# B&R Automation Studio project dbserv_0640 (part 19)

#### iodrv.c
```c
#ifdef _DEFAULT_INCLUDES
	#include <AsDefault.h>
#endif
/******************************************************************************
*    COPYRIGHT    BERNECKER + RAINER Industrie-Elektronik Ges.m.b.H           *
*******************************************************************************
*  Projekt:  I/O-Treiber
*  Teil:     Hauptprogramm
*  Datei:    iodrv.c
*  Typ:      GNU-C (32 Bit)
*------------------------------------------------------------------------------
*  Revision: 01.00
*  Datum:    05-04-2006
*  Autor:    WAI
*------------------------------------------------------------------------------
*  Funktion:
*------------------------------------------------------------------------------
*  Rev.  | Datum    | Name | Kommentar
*  ------+----------+------+---------------------------------------------------
*  01.00 | 05-04-06 | WAI  | Datei-Erstellung
*  01.01 | 26-11-10 | WAI  | Schreibzugriff auf PVs aktiviert
*        |          |      |
******************************************************************************/

/***********************************************************************/
/* Headerfiles einbinden                                               */
/***********************************************************************/

#include <bur\plc.h>			/* RPS-spezifische Typendeklarationen */
#include <string.h>
#include <dvframe.h>
#include <sys_lib.h>
#include <brsystem.h>
#include <fileio.h>
#include "iodrv.h"				/* globale Variablen und Konstanten */
#include "iodrv_parse.h"		/* Parser Funktionen */
#include "dbserv.h"				/* Meldeserver */

_LOCAL_RETAIN	BOOL	go	;
_LOCAL	UINT	LinkStat,SetStat,ScanStat,GetStat;

/***********************************************************************/
/* 					Initialisierungs-Unterprogramm                     */
/***********************************************************************/

void _INIT init_iodrv(void)
{

	int	item,i;
	IODRV_DP_Info_typ		*pIODRV_DP_Info;

	/*--------------------------------*/
	/* Variablen initialisieren       */
	/*--------------------------------*/
	for(i=0;i<ITEM_DIAGNOSE_SIZE;i++) {
		IODRV_ItemDiagnose[i].showData	= 0;
	}

	memset(&SYS_Statistic,0,sizeof(SYS_Statistic));

	myidBrServer			= 0;											/* ID BR-Server */

	rt_info.enable = 1; 													/* Taskklassenzykluszeit ermitteln */
	RTInfo(&rt_info);
	if(rt_info.status==0)	CycleTime	= (rt_info.cycle_time / 1000);		/* Zykluszeit in ms */
	else 					CycleTime	= 10;								/* Zykluszeit in ms */

	Error	= 0;															/* Generelle Variable fuer Initialisierungsfehler */

	initPAB = 1;

	/*****************************************************************************/
	/* Initialisierung nach Konfigurationsdatenmodul dplist und typlist (DbServ) */
	/*****************************************************************************/

	/*--------------------------------------------------*/
	/* Konfiguration aus Konfigurationsmodulen auslesen */
	/*--------------------------------------------------*/

	iodrv_parser();

	/* Kein Schwerwiegender Fehler beim Parsen */
	if(IODRV_ParserInfo.error==0) {
		/* für alle Items die PV suchen */
		for(item=0;item<IODRV_ParserInfo.NrOfItems;item++)	{
			pIODRV_DP_Info = (IODRV_DP_Info_typ *) (IODRV_ParserInfo.memAdr);
			pIODRV_DP_Info += item;

			if(pIODRV_DP_Info->DPNameLen && pIODRV_DP_Info->DPName !=NULL)	{
				/* PV-Namen aus DP- und Item-Namen zusammensetzen */
				strncpy(pIODRV_DP_Info->PVName,pIODRV_DP_Info->DPName,pIODRV_DP_Info->DPNameLen);
				if(pIODRV_DP_Info->ItemNameLen && pIODRV_DP_Info->ItemName !=NULL)	{
					strncat(pIODRV_DP_Info->PVName,pIODRV_DP_Info->ItemName,pIODRV_DP_Info->ItemNameLen);
				}
				/* PV-Adresse bestimmen */
				statePV_xgetadr = PV_xgetadr(pIODRV_DP_Info->PVName, &pIODRV_DP_Info->PVAdrs, &pIODRV_DP_Info->PVDataLen);
				if (statePV_xgetadr != 0) {
					/* Fehler PV */
						iodrv_parser_warn(PARS_ERR_PV_NOT_FOUND,"PV nicht vorhanden", pIODRV_DP_Info->PVName, 0,0, 0, 0, 0, 0);
				}
			}
		}
	}
}
/************************************************************************/
/* schreibt aktuellen Datenpunkt in das PAB 							*/
void WritePVtoPAB(IODRV_DP_Info_typ *pIODRV_DP_Info)
{
	int						do_it;
	PAR_TYPE				WertServer;
	UDINT					SizeServer;

	/* nur Lese- bzw. Schreib/Lese-Items an das PAB übergeben */
	if (myidBrServer == 0) {
		pIODRV_DP_Info->ErrorInfo = 2;				/* Info Server ID unbekannt */
	}
	else {
		pIODRV_DP_Info->AccessCounter += 1;			/* Zaehler inkrementieren: Signal wird an Server uebergeben */
		do_it = 1;

		switch(pIODRV_DP_Info->ItemTypNr) {
			case BOOL_IDX:
				pIODRV_DP_Info->ValueIO = *(BOOL *) pIODRV_DP_Info->PVAdrs;
				SizeServer  = sizeof(BOOL);
				if(pIODRV_DP_Info->Invers)	{
					WertServer.b	= (BOOL)pIODRV_DP_Info->ValueIO ^1;
				}
				else {
					WertServer.b	= (BOOL)pIODRV_DP_Info->ValueIO;
				}
				if(!initPAB && !WertServer.b && pIODRV_DP_Info->Quitt)	{
					do_it = 0;				/* gegangener, quittierpflichtiger DP nicht in PAB eintragen */
				}
				break;
			case USINT_IDX:
				WertServer.ui1	= *(USINT*)	pIODRV_DP_Info->PVAdrs;
				SizeServer  = sizeof(USINT);
				break;
			case SINT_IDX:
				WertServer.i1	= *(SINT*)	pIODRV_DP_Info->PVAdrs;
				SizeServer  = sizeof(SINT);
				break;
			case UINT_IDX:
				WertServer.ui2	= *(UINT*)	pIODRV_DP_Info->PVAdrs;
				SizeServer  = sizeof(UINT);
				break;
			case INT_IDX:
				WertServer.i2	= *(INT*)	pIODRV_DP_Info->PVAdrs;
				SizeServer  = sizeof(INT);
				break;
			case UDINT_IDX:
				WertServer.ui4	= *(UDINT*)	pIODRV_DP_Info->PVAdrs;
				SizeServer  = sizeof(UDINT);
				break;
			case DINT_IDX:
				WertServer.i4	= *(DINT*)	pIODRV_DP_Info->PVAdrs;
				SizeServer  = sizeof(DINT);
				break;
			default:
				WertServer.i2	= *(INT*)	pIODRV_DP_Info->PVAdrs;
				SizeServer  = sizeof(INT);
				break;
		}
		if(do_it)	{
			StatusSetValueItem = SetValueItem ((ACCESS_SERVER*)	myidBrServer,
												pIODRV_DP_Info->AnlagenNr,
												1,									/* Stationsnummer  immer 1 */
												pIODRV_DP_Info->DPTypNr,	  		/* Datenpunkttyp    */
												pIODRV_DP_Info->DPNr,			 	/* Datenpunktnummer */
												pIODRV_DP_Info->ItemNr,				/* Item */
												(USINT *) &WertServer,				/* Adresse Messwert */
												SizeServer,
												TimeBuf,
												0,			/* TimeStampNow=0 wegen Alarmliste, setze Zeitstempel bei Bedarf */
												1);
			if(!StatusSetValueItem)	{
				pIODRV_DP_Info->AccessCounter += 1;				/* Zaehler inkrementieren: Uebergabe an Server korrekt erfolgt */
				pIODRV_DP_Info->ErrorInfo		= 0;
			}
			else {
				pIODRV_DP_Info->ErrorInfo = 3;
			}
		}
	}
}

/***********************************************************************/
/* 						zyklisches Hauptprogramm                       */
/***********************************************************************/

void _CYCLIC cyclic_iodrv(void)
{
	int						item;
	IODRV_DP_Info_typ		*pIODRV_DP_Info;
	USINT	WriteBuffer[32];
	UDINT	len, lenTimeStamp;
	USINT	*pByteValue;

	/* Einlesen der Echtzeituhr */
	RTC_gettime(&TimeBuf);

	/* ID Meldeserver besorgen */
	get_idBrServer();

	if(go)	{
		go=0;
		iodrv_parser();

		/* Kein Schwerwiegender Fehler beim Parsen */
		if(IODRV_ParserInfo.error==0) {
			/* für alle Items die PV suchen */
			for(item=0;item<IODRV_ParserInfo.NrOfItems;item++)	{
				pIODRV_DP_Info = (IODRV_DP_Info_typ *) (IODRV_ParserInfo.memAdr);
				pIODRV_DP_Info += item;

				if(pIODRV_DP_Info->DPNameLen && pIODRV_DP_Info->DPName !=NULL)	{
					/* PV-Namen aus DP- und Item-Namen zusammensetzen */
					strncpy(pIODRV_DP_Info->PVName,pIODRV_DP_Info->DPName,pIODRV_DP_Info->DPNameLen);
					if(pIODRV_DP_Info->ItemNameLen && pIODRV_DP_Info->ItemName !=NULL)	{
						strncat(pIODRV_DP_Info->PVName,pIODRV_DP_Info->ItemName,pIODRV_DP_Info->ItemNameLen);
					}
					/* PV-Adresse bestimmen */
					statePV_xgetadr = PV_xgetadr(pIODRV_DP_Info->PVName, &pIODRV_DP_Info->PVAdrs, &pIODRV_DP_Info->PVDataLen);
					if (statePV_xgetadr != 0) {
						/* Fehler PV */
						iodrv_parser_warn(PARS_ERR_PV_NOT_FOUND,"PV nicht vorhanden", pIODRV_DP_Info->PVName, 0,0, 0, 0, 0, 0);
					}
				}
			}
		}
	}

	/* Diagnose */
	iodrv_mem_diagnose();

	/* -------------------------------*/
	/* Uebergabe an Server            */
	/* -------------------------------*/

	for(item=0;item<IODRV_ParserInfo.NrOfItems;item++)	{
		pIODRV_DP_Info = (IODRV_DP_Info_typ *) (IODRV_ParserInfo.memAdr);
		pIODRV_DP_Info += item;

		if(pIODRV_DP_Info->PVAdrs != NULL)	{
			if(pIODRV_DP_Info->Dir == cKW_READ)	{
				WritePVtoPAB(pIODRV_DP_Info);				/* PV ins PAB schreiben */
			}
			else if(pIODRV_DP_Info->Dir == cKW_READWRITE || pIODRV_DP_Info->Dir == cKW_WRITE)	{
				/* Item zum Schreiben anmelden */
				LinkStat = LinkWriteItem((ACCESS_SERVER*)myidBrServer, cINSTANCE_IODRV,
						pIODRV_DP_Info->AnlagenNr, 1, pIODRV_DP_Info->DPTypNr, pIODRV_DP_Info->DPNr, pIODRV_DP_Info->ItemNr,
						(UDINT)pIODRV_DP_Info);
				if (LinkStat != cEC_OK && LinkStat != cEC_ITEM_ALREADY_LINKED)	pIODRV_DP_Info->ErrorInfo = LinkStat;
				/* prüfen, ob Item geschrieben wurde */
				ScanStat = ScanWriteItem((ACCESS_SERVER*)myidBrServer, cINSTANCE_IODRV,
											WriteBuffer, sizeof(WriteBuffer),
											&len, &lenTimeStamp);
				if (ScanStat != cEC_OK)	pIODRV_DP_Info->ErrorInfo = ScanStat;
				if (ScanStat == cEC_OK) {
					/* für mich ? */
					GetStat = cEC_NO_DATA_IN_WRITEBUFFER;
					if (((WRITE_PIPE_DATA*)WriteBuffer)->pData == (unsigned char *)pIODRV_DP_Info) {
						GetStat = GetWriteItem((ACCESS_SERVER*)myidBrServer, cINSTANCE_IODRV,
												WriteBuffer, sizeof(WriteBuffer),
												&len, &lenTimeStamp);
						if (GetStat != cEC_OK)	pIODRV_DP_Info->ErrorInfo = GetStat;
						if (GetStat== cEC_OK) {
							if (((WRITE_PIPE_DATA*)WriteBuffer)->length == pIODRV_DP_Info->PVDataLen) {
								pByteValue = WriteBuffer + sizeof(WRITE_PIPE_DATA);
/* #if 0 26.11.10 Wai Kommentar entfernt */
								switch(pIODRV_DP_Info->ItemTypNr) {
									case BOOL_IDX:
										*(BOOL *)pIODRV_DP_Info->PVAdrs =  *(BOOL*)pByteValue;
										break;
									case USINT_IDX:
										*(USINT *)pIODRV_DP_Info->PVAdrs =  *(USINT*)pByteValue;
										break;
									case SINT_IDX:
										*(SINT *)pIODRV_DP_Info->PVAdrs =  *(SINT*)pByteValue;
										break;
									case UINT_IDX:
										*(UINT *)pIODRV_DP_Info->PVAdrs =  *(UINT*)pByteValue;
										break;
									case INT_IDX:
										*(INT *)pIODRV_DP_Info->PVAdrs =  *(INT*)pByteValue;
										break;
									case UDINT_IDX:
										*(UDINT *)pIODRV_DP_Info->PVAdrs =  *(UDINT*)pByteValue;
										break;
									case DINT_IDX:
										*(DINT *)pIODRV_DP_Info->PVAdrs =  *(DINT*)pByteValue;
										break;
								}
/* #endif 26.11.10 Wai Kommentar entfernt */

								/* Wert auch nach PAB zurückschreiben */
								SetStat = SetValueItem((ACCESS_SERVER*)myidBrServer,
										pIODRV_DP_Info->AnlagenNr, 1, pIODRV_DP_Info->DPTypNr, pIODRV_DP_Info->DPNr, pIODRV_DP_Info->ItemNr,
										pByteValue, sizeof(INT), TimeBuf, 0, TRUE);
								if (SetStat != cEC_OK)	pIODRV_DP_Info->ErrorInfo = SetStat;
							} /* (((WRITE_PIPE_DATA*)WriteBuffer)->length == PVDataLen */
							else {
								SetStat = cEC_INVALID_LENGTH;
								if (SetStat != cEC_OK)	pIODRV_DP_Info->ErrorInfo = SetStat;
							}
						} /* (intStat == cEC_OK) */
					} /* (((WRITE_PIPE_DATA*)WriteBuffer)->pData == (unsigned char*)inst->FubRef.this) */
				} /* (intStat == cEC_OK) */
				if (ScanStat != cEC_OK || GetStat != cEC_OK)	{
					/* keine Schreibdaten vorhanden: PV ins PAB schreiben */
					if(pIODRV_DP_Info->Dir == cKW_READWRITE)	{
						WritePVtoPAB(pIODRV_DP_Info);				/* PV ins PAB schreiben */
					}
				}
			} /* else if(pIODRV_DP_Info->Dir == cKW_READWRITE || pIODRV_DP_Info->Dir == cKW_WRITE)	*/
		} /* if(pIODRV_DP_Info->PVAdrs != NULL)	*/
	} /* for all Items */
	if(myidBrServer) initPAB = 0;

}

/*** eof *****************************************************************************/
```

#### iodrv_parse.c
```c
#ifdef _DEFAULT_INCLUDES
	#include <AsDefault.h>
#endif
/******************************************************************************
*    COPYRIGHT    BERNECKER + RAINER Industrie-Elektronik Ges.m.b.H           *
*******************************************************************************
*  Projekt:  I/O-Treiber
*  Teil:     Parserfunktionen
*  Datei:    iodrv_parse.c
*  Typ:      GNU-C (32 Bit)
*------------------------------------------------------------------------------
*  Revision: 01.00
*  Datum:    05-04-2006
*  Autor:    WAI
*------------------------------------------------------------------------------
*  Funktion:
*------------------------------------------------------------------------------
*  Rev.  | Datum    | Name | Kommentar
*  ------+----------+------+---------------------------------------------------
*  01.00 | 05-04-06 | WAI  | Datei-Erstellung
*  02.00 | 10-07-26 | BIE  | strnicmp gegen strncasecmp ersetzt
*        |          |      |
******************************************************************************/
#include <bur\plc.h>			/* RPS-spezifische Typendeklarationen */
#include <string.h>
#include <dvframe.h>
#include <sys_lib.h>
#include <asbrstr.h>
#include <brsystem.h>
#include "iodrv.h"
#include "iodrv_parse.h"
#include "parser.h"

/**********************************************************
*		Konfiguration aus Datenmodul auslesen
**********************************************************/
void iodrv_parser()
{
	plcbit				BlockFound,DPFound,TypFound,ItemFound;
	IODRV_DP_Info_typ		*pIODRV_DP_Info;
	unsigned char ANr[20];

	memset(&IODRV_ParserInfo,0,sizeof(IODRV_ParserInfo));
	IODRV_ParserInfo.ErrorMsg = 1;									/* Freigabe: Fehlermeldungen ins Logbuch eintragen */

	/*--------------------------------------------------*/
	/* Info ueber Datenmodul dplist und typlist besorgen*/
	/*--------------------------------------------------*/

	DOI_dplist.enable	= 1;
	DOI_dplist.pName	= (unsigned long) DATA_OBJEKT_DPLIST;
	DatObjInfo((DatObjInfo_typ*) &DOI_dplist);

	DOI_typlist.enable	= 1;
	DOI_typlist.pName	= (unsigned long) DATA_OBJEKT_TYPLIST;
	DatObjInfo((DatObjInfo_typ*) &DOI_typlist);

	/*--------------------------------------------------*/
	/* Fehlermeldung: Datenmodul dplist nicht vorhanden */
	/*--------------------------------------------------*/
	if(DOI_typlist.status) {
		iodrv_parser_err(PARS_ERR_DPLIST_NOT_FOUND, "Datenmodul fehlt:", (unsigned char *) DOI_dplist.pName, 0, 0, 0, 0, 0, 0);
	}

	/*--------------------------------------------------*/
	/* Fehlermeldung: Datenmodul typlist nicht vorhanden */
	/*--------------------------------------------------*/
	if(DOI_typlist.status) {
		iodrv_parser_err(PARS_ERR_TYPLIST_NOT_FOUND, "Datenmodul fehlt:", (unsigned char *) DOI_typlist.pName, 0, 0, 0, 0, 0, 0);
	}

	/*--------------------------------------------------*/
	/* Globale Parameter lesen							*/
	/*--------------------------------------------------*/
	if(!IODRV_ParserInfo.error) {

		iodrv_parser_dplist_clear();									/* Parsen von Beginn an */

		memset(&IODRV_GlobalData,0,sizeof(IODRV_GlobalData));			/* Parameterstruktur loeschen */

		iodrv_parser_global();											/* Parameter parsen */
	}

	/*------------------------------------------------------*/
	/* Anzahl Datenpunkte und Items ermitteln				*/
	/*------------------------------------------------------*/

	if(!IODRV_ParserInfo.error) {

		IODRV_ParserInfo.ErrorMsg = 0;															/* Keine Eintrage ins Logbuch */
		iodrv_parser_dplist_clear();															/* dplist von Beginn an Parsen */
		memset(&IODRV_BlockData,0,sizeof(IODRV_BlockData));										/* Info ueber Blockparameter loeschen */

		do {
			memset(&IODRV_DPData,0,sizeof(IODRV_DPData));											/* Info ueber Datenpunkt loeschen */
			copyItemData((IODRV_ItemData_typ *) &IODRV_DPData,(IODRV_ItemData_typ *) &IODRV_BlockData);	/* Blockparameter uebernehmen */

			BlockFound	= 0;
			DPFound		= 0;

			iodrv_parser_dpinfo((plcbit *) &BlockFound,(plcbit *) &DPFound);						/* Nächsten Datenpunkt für IODRV-Treiber suchen */

			if(DPFound) {																	/* Datenpunkt für IODRV-Treiber gefunden */
				IODRV_ParserInfo.NrOfDataPoints++;											/* Anzahl Datenpunkte pro Linie zählen */
				if(IODRV_DPData.Typ.defined) {												/* Ist zu dem Datenpunkt der Datentyp definiert ? */
					iodrv_parser_typlist_clear();											/* typlist von Beginn an Parsen */
					TypFound = iodrv_parser_dptype(IODRV_DPData.Typ.name, IODRV_DPData.Typ.size); /* Datentyp in typlist suchen */
					if(TypFound) {															/* Datentyp wurde in typlist gefunden */
						/* Anzahl Items des Datenpunktes ermitteln */
						do {
							memset(&IODRV_ItemData,0,sizeof(IODRV_ItemData));				/* Struktur für ITEM-Parameter loeschen */
							ItemFound = iodrv_parser_iteminfo();							/* Item in typlist suchen */
							if(ItemFound) {													/* Item wurde gefunden */
								copyItemData((IODRV_ItemData_typ *) &IODRV_ItemData,(IODRV_ItemData_typ *) &IODRV_DPData);
								IODRV_ParserInfo.NrOfItems++;								/* Anzahl der Items ermitteln */
							}
						} while(ItemFound);

					} /* if(TypFound) */
				} /* if(IODRV_DPData.Typ.defined) */
			} /* if(DPFound) */
		} while(DPFound || BlockFound);
	} /* if(!IODRV_ParserInfo.error) */

	/*------------------------------------------------------*/
	/* Speicher fuer alle Items allokieren					*/
	/*------------------------------------------------------*/

	if(!IODRV_ParserInfo.error) {
		IODRV_ParserInfo.ErrorMsg	= 1;					/* Freigabe: Fehlermeldungen ins Logbuch eintragen */
		IODRV_ParserInfo.memSize = IODRV_ParserInfo.NrOfItems * sizeof(IODRV_DP_Info_typ);
		IODRV_ParserInfo.allocStatus = TMP_alloc(IODRV_ParserInfo.memSize, (void**) &IODRV_ParserInfo.memAdr); 	/* allocate new memory from RAM*/
		if(IODRV_ParserInfo.allocStatus) {
			iodrv_parser_err(PARS_ERR_MEM_ALLOC, "Fehler TMP_alloc:", 0, "Groesse:", IODRV_ParserInfo.memSize, "Status:", (long) IODRV_ParserInfo.allocStatus, 0, 0);
		}
		else {
			memset((void *) IODRV_ParserInfo.memAdr,0,IODRV_ParserInfo.memSize);
		}
	}

	/*-----------------------------------------------------------------------*/
	/* Iteminformationen auslesen und in Speicher eintragen     */
	/*-----------------------------------------------------------------------*/

	if(!IODRV_ParserInfo.error) {

		iodrv_parser_dplist_clear();																/* dplist von Beginn an Parsen */
		memset(&IODRV_BlockData,0,sizeof(IODRV_BlockData));											/* Info ueber Blockparameter loeschen */

		do {
			memset(&IODRV_DPData,0,sizeof(IODRV_DPData));											/* Info ueber Datenpunkt loeschen */
			copyItemData((IODRV_ItemData_typ *) &IODRV_DPData,(IODRV_ItemData_typ *) &IODRV_BlockData);	/* Blockparameter uebernehmen */
			BlockFound	= 0;
			DPFound		= 0;
			iodrv_parser_dpinfo((plcbit *) &BlockFound,(plcbit *) &DPFound);						/* Nächsten Datenpunkt für IODRV-Treiber suchen */
			if(DPFound) {																		/* Datenpunkt für IODRV-Treiber gefunden */
				if(iodrv_parser_dpinfo_ok((IODRV_ItemData_typ *) &IODRV_DPData)) {					/* Alle notwendigen Angaben vorhanden und korrekt ? */
																								/* Zugehoerigen Linienindex suchen */
					iodrv_parser_typlist_clear();												/* typlist von Beginn an Parsen */
					TypFound = iodrv_parser_dptype(IODRV_DPData.Typ.name, IODRV_DPData.Typ.size); /* Datentyp in typlist suchen */
					if(TypFound) {															/* Datentyp wurde in typlist gefunden */
						/* Anzahl Items des Datenpunktes ermitteln */
						do {
							memset(&IODRV_ItemData,0,sizeof(IODRV_ItemData));					/* Struktur für ITEM-Parameter loeschen */
																								/* Parameter des Datenpunktes auf Item übertragen */
							copyItemData((IODRV_ItemData_typ *) &IODRV_ItemData,(IODRV_ItemData_typ *) &IODRV_DPData);

							ItemFound = iodrv_parser_iteminfo();								/* Item in typlist suchen */
							if(ItemFound) {													/* Item wurde gefunden */

																							/* Pruefen, ob Parameter vollstaendig und korrekt sind */
								if(iodrv_parser_iteminfo_ok((IODRV_ItemData_typ *) &IODRV_ItemData)) {
									pIODRV_DP_Info = (IODRV_DP_Info_typ *) (IODRV_ParserInfo.memAdr);
									pIODRV_DP_Info += IODRV_ParserInfo.ActItemIdx;

																						/* Daten in Speicher eintragen */
									pIODRV_DP_Info->AnlagenNr	= (UINT)	IODRV_ItemData.AnlagenNr.value;
									pIODRV_DP_Info->DPNr		= (UINT)	IODRV_ItemData.DPNr.value;
									pIODRV_DP_Info->DPTypNr		= (UINT)	IODRV_ItemData.DPTypNr.value;
									pIODRV_DP_Info->DPName		= (USINT *)	IODRV_ItemData.DPName.name;
									pIODRV_DP_Info->DPNameLen	= (UINT)	IODRV_ItemData.DPName.size;
									pIODRV_DP_Info->ItemNr		= (UINT)	IODRV_ItemData.ItemNr.value;
									pIODRV_DP_Info->ItemTypNr	= (USINT)	IODRV_ItemData.ItemTypNr.value;
									pIODRV_DP_Info->ItemName	= (USINT *)	IODRV_ItemData.ItemName.name;
									pIODRV_DP_Info->ItemNameLen	= (UINT)	IODRV_ItemData.ItemName.size;
									pIODRV_DP_Info->Invers		= (USINT)	IODRV_ItemData.Invers.value;
									pIODRV_DP_Info->Quitt		= (USINT)	IODRV_ItemData.Quitt.value;
									pIODRV_DP_Info->Dir			= (USINT)	IODRV_ItemData.Dir.value;

									IODRV_ParserInfo.ActItemIdx++;
								} /* if(!error) */
							} /* if(!error) */
						} while(ItemFound);
					} /* if(TypFound) */
				} /* if(iodrv_parser_dpinfo_ok())*/
			} /* if(DPFound) */
		} while(DPFound || BlockFound);
	} /* if(!IODRV_ParserInfo.error) */

	strcpy(MsgTxt,ERR_MSG_PRE_STRG);
	strcat(MsgTxt," Parser beendet");
	ERRxwarning( 0, bin_to_bcd_8(0),MsgTxt);

	strcpy(MsgTxt,ERR_MSG_PRE_STRG);
	strcat(MsgTxt," Anzahl Meldungen ");
	brsitoa(IODRV_ParserInfo.NrOfLogEntrys, (UDINT) &ANr);
	strcat(MsgTxt,ANr);
	ERRxwarning( 0, bin_to_bcd_8((unsigned long) IODRV_ParserInfo.NrOfLogEntrys), MsgTxt);

}

/**********************************************************
*		Globale Parameter aus Datennmodul lesen
**********************************************************/
void iodrv_parser_global()
{

	BOOL			dataReady;

		/* ----------------------------------------- */
	 	/* Globale Eintraege fuer IODRV-Treiber parsen */
		/* ----------------------------------------- */

		/* Parser-Status loeschen */
		State_find_StationTypPoint	= 0;
		State_find_Section			= 0;
		State_find_Data				= 0;

		while (PaDPList.pParser < (unsigned char*) DOI_dplist.pDatObjMem + DOI_dplist.len) {

			/* Suche nach Stations/Typ/Punkt-Beschreibung */
			State_find_StationTypPoint = find_StationTypPoint (	(unsigned char*) DOI_dplist.pDatObjMem, PaDPList.pParser,
																(unsigned char*) DOI_dplist.pDatObjMem + DOI_dplist.len,
																&PaDPList.pParser, &PaDPList.pParserLine, &PaDPList.pParserErr, &PaDPList.CountLines,
																&PaDPList.pDataArg1, &PaDPList.SizeArg1,
																&PaDPList.pDataArg2, &PaDPList.SizeArg2,
																&PaDPList.SectionType);
			/* keine Daten oder Fehler aufgetreten ? */
			if (State_find_StationTypPoint < 0) {
				break;
			}

			/* Pointer auf Station/Typ/Punkt */
			switch (PaDPList.SectionType) {

				/* ------------------ */
				/* Stations-Abschnitt */
				/* ------------------ */
				case cCD_STATION:
					do {
						State_find_Section = find_Section (
							(unsigned char*) DOI_dplist.pDatObjMem, PaDPList.pParser,
															(unsigned char*) DOI_dplist.pDatObjMem + DOI_dplist.len,
															&PaDPList.pParser, &PaDPList.pParserLine, &PaDPList.pParserErr, &PaDPList.CountLines,
															&PaDPList.pDataArg1, &PaDPList.SizeArg1,
															&PaDPList.pDataArg2, &PaDPList.SizeArg2,
															KW_IODRV_SECTION);

						/* keine Daten oder Fehler aufgetreten ? */
						if (State_find_Section < 0) {
							break;
						}

						/* Pointer auf Anfang der Sektion stellen */
						if (PaDPList.pDataArg2 != NULL) {
							PaDPList.pParser = PaDPList.pDataArg2;
						}
						else {
							continue;
						}

						/* alle Daten der Sektion bearbeiten */
						dataReady	= 0;
						do {
							/* Daten der Sektion anfordern */
							State_find_Data = find_Data (	(unsigned char*) DOI_dplist.pDatObjMem, PaDPList.pParser,
															(unsigned char*) DOI_dplist.pDatObjMem + DOI_dplist.len,
															  &PaDPList.pParser, &PaDPList.pParserLine, &PaDPList.pParserErr, NULL,
															  &PaDPList.pDataArg1, &PaDPList.SizeArg1,
															  &PaDPList.pDataArg2, &PaDPList.SizeArg2,
															  &PaDPList.pDataArg3, &PaDPList.SizeArg3);

							/* Zeilenende erreicht */
							if (State_find_Data == -1) {
								PaDPList.pParser++;
							}
							/* Daten vorhanden */
							else if (State_find_Data == TRUE) {
								/* noch keine globalen Daten vorhanden */
								if (0) {
								}
								/* Unbekannter Eintrag */
								else {
									iodrv_parser_warn(PARS_ERR_UNKNOWN_GLOBAL_ENTRY,"Eintrag unbekannt:", PaDPList.pParserLine, " / Zeile =", (long) PaDPList.CountLines, 0, 0, 0, 0);
								}
							}

							/* Endebedinung der Schleife: Keine Daten mehr vorhanden, oder Ende des Datenmodules erreicht */
							if((State_find_Data!=TRUE) && (State_find_Data!=-1))					dataReady = 1;
							if(PaDPList.pParser >= (unsigned char*) DOI_dplist.pDatObjMem + DOI_dplist.len)	dataReady = 1;
						} while (!dataReady);
					} while (State_find_Section == TRUE);
					break;
				case cCD_TYP:
					break;
				case cCD_POINT:
					break;
			}
		}
}

/*****************************************************************
*		Informationen ueber einen Datenpunkt ermitteln
******************************************************************/
void iodrv_parser_dpinfo(plcbit *pBlockFound, plcbit *pDPFound)
{

		*pDPFound	= 0;
		*pBlockFound= 0;

		/* -------------------------------------------- */
	 	/* Datenpunkt Eintraege fuer IODRV-Treiber parsen */
		/* -------------------------------------------- */

		/* Parser-Status loeschen */
		State_find_StationTypPoint	= 0;
		State_find_Section			= 0;
		State_find_Data				= 0;

		while (!*pDPFound && !*pBlockFound && (PaDPList.pParser < (unsigned char*) DOI_dplist.pDatObjMem + DOI_dplist.len)) {

			/* Suche nach Stations/Typ/Punkt-Beschreibung */
			State_find_StationTypPoint = find_StationTypPoint (	(unsigned char*) DOI_dplist.pDatObjMem, PaDPList.pParser,
																(unsigned char*) DOI_dplist.pDatObjMem + DOI_dplist.len,
																&PaDPList.pParser, &PaDPList.pParserLine, &PaDPList.pParserErr, &PaDPList.CountLines,
																&PaDPList.pDataArg1, &PaDPList.SizeArg1,
																&PaDPList.pDataArg2, &PaDPList.SizeArg2,
																&PaDPList.SectionType);
			/* keine Daten oder Fehler aufgetreten ? */
			if (State_find_StationTypPoint < 0) {
				break;
			}

			/* Pointer auf Station/Typ/Punkt */
			switch (PaDPList.SectionType) {
				/* ------------------ */
				/* Datentyp-Abschnitt */
				/* ------------------ */
				case cCD_POINT:

					/* Parserposition zwischenspeichern */
					memcpy(&PaDPListSave,&PaDPList,sizeof(PaDPListSave));

					pPointName = PaDPList.pDataArg1, lenPointName = PaDPList.SizeArg1;

					/* Suchen nach Sektion "IODRV" */
					do {
						State_find_Section = find_Section (	(unsigned char*) DOI_dplist.pDatObjMem, PaDPList.pParser,
															(unsigned char*) DOI_dplist.pDatObjMem + DOI_dplist.len,
															&PaDPList.pParser, 	 &PaDPList.pParserLine, &PaDPList.pParserErr, &PaDPList.CountLines,
															&PaDPList.pDataArg1, &PaDPList.SizeArg1,
															&PaDPList.pDataArg2, &PaDPList.SizeArg2,
															KW_IODRV_SECTION);

						/* keine Daten oder Fehler aufgetreten ? */
						if (State_find_Section < 0) {
							break;
						}

						/* Pointer auf Anfang der Sektion stellen */
						if (PaDPList.pDataArg2 != NULL) {
							PaDPList.pParser = PaDPList.pDataArg2;
						}
						else {
							continue;
						}

						/* alle Daten der Sektion bearbeiten */

						IODRV_DPData.DPName.name = pPointName;
						IODRV_DPData.DPName.size = lenPointName;
						IODRV_DPData.DPName.defined = 1;

						*pDPFound		= 1;
						iodrv_parser_data((unsigned char*) DOI_dplist.pDatObjMem,
										(unsigned char*) DOI_dplist.pDatObjMem + DOI_dplist.len,
										(Parser_typ *) &PaDPList,
										(IODRV_ItemData_typ *) &IODRV_DPData,
										IODRV_SECTION,DP_PART);

					} while (State_find_Section == TRUE);

					/* Parserposition rückholen */
					memcpy(&PaDPList,&PaDPListSave,sizeof(PaDPList));

					/* Suchen nach Sektion "ALL" */
					do {
						State_find_Section = find_Section (	(unsigned char*) DOI_dplist.pDatObjMem, PaDPList.pParser,
															(unsigned char*) DOI_dplist.pDatObjMem + DOI_dplist.len,
															&PaDPList.pParser, &PaDPList.pParserLine, &PaDPList.pParserErr, &PaDPList.CountLines,
															&PaDPList.pDataArg1, &PaDPList.SizeArg1,
															&PaDPList.pDataArg2, &PaDPList.SizeArg2,
															KW_ALL_SECTION);

						/* keine Daten oder Fehler aufgetreten ? */
						if (State_find_Section < 0) {
							break;
						}

						/* Pointer auf Anfang der Sektion stellen */
						if (PaDPList.pDataArg2 != NULL) {
							PaDPList.pParser = PaDPList.pDataArg2;
						}
						else {
							continue;
						}

						/* alle Daten der Sektion bearbeiten */
						iodrv_parser_data((unsigned char*) DOI_dplist.pDatObjMem,
										(unsigned char*) DOI_dplist.pDatObjMem + DOI_dplist.len,
										(Parser_typ *) &PaDPList,
										(IODRV_ItemData_typ *) &IODRV_DPData,
										ALL_SECTION,DP_PART);

					} while (State_find_Section == TRUE);
					break;

				/* ------------------ */
				/* Block-Abschnitt    */
				/* ------------------ */
				case cCD_TYP:
					if(strncasecmp(PaDPList.pDataArg1, KW_BLOCK_SECTION, PaDPList.SizeArg1) == 0 && strlen(KW_BLOCK_SECTION) == PaDPList.SizeArg1 ) {
						*pBlockFound = 1;

						/* Parserposition zwischenspeichern */
						memcpy(&PaDPListSave,&PaDPList,sizeof(PaDPListSave));

						/* Suchen nach Sektion "IODRV" */
						do {
							State_find_Section = find_Section (	(unsigned char*) DOI_dplist.pDatObjMem, PaDPList.pParser,
																(unsigned char*) DOI_dplist.pDatObjMem + DOI_dplist.len,
																&PaDPList.pParser, 	 &PaDPList.pParserLine, &PaDPList.pParserErr, &PaDPList.CountLines,
																&PaDPList.pDataArg1, &PaDPList.SizeArg1,
																&PaDPList.pDataArg2, &PaDPList.SizeArg2,
																KW_IODRV_SECTION);

							/* keine Daten oder Fehler aufgetreten ? */
							if (State_find_Section < 0) {
								break;
							}

							/* Pointer auf Anfang der Sektion stellen */
							if (PaDPList.pDataArg2 != NULL) {
								PaDPList.pParser = PaDPList.pDataArg2;
							}
							else {
								continue;
							}

							/* alle Daten der Sektion bearbeiten */

							iodrv_parser_data((unsigned char*) DOI_dplist.pDatObjMem,
											(unsigned char*) DOI_dplist.pDatObjMem + DOI_dplist.len,
											(Parser_typ *) &PaDPList,
											(IODRV_ItemData_typ *) &IODRV_BlockData,
											IODRV_SECTION,DP_PART);

						} while (State_find_Section == TRUE);

						/* Parserposition rückholen */
						memcpy(&PaDPList,&PaDPListSave,sizeof(PaDPList));

						/* Suchen nach Sektion "ALL" */
						do {
							State_find_Section = find_Section (	(unsigned char*) DOI_dplist.pDatObjMem, PaDPList.pParser,
																(unsigned char*) DOI_dplist.pDatObjMem + DOI_dplist.len,
																&PaDPList.pParser, &PaDPList.pParserLine, &PaDPList.pParserErr, &PaDPList.CountLines,
																&PaDPList.pDataArg1, &PaDPList.SizeArg1,
																&PaDPList.pDataArg2, &PaDPList.SizeArg2,
																KW_ALL_SECTION);

							/* keine Daten oder Fehler aufgetreten ? */
							if (State_find_Section < 0) {
								break;
							}

							/* Pointer auf Anfang der Sektion stellen */
							if (PaDPList.pDataArg2 != NULL) {
								PaDPList.pParser = PaDPList.pDataArg2;
							}
							else {
								continue;
							}

							/* alle Daten der Sektion bearbeiten */
							iodrv_parser_data((unsigned char*) DOI_dplist.pDatObjMem,
											(unsigned char*) DOI_dplist.pDatObjMem + DOI_dplist.len,
											(Parser_typ *) &PaDPList,
											(IODRV_ItemData_typ *) &IODRV_BlockData,
											ALL_SECTION,DP_PART);

						} while (State_find_Section == TRUE);
					}
					break;

			}
		}
}

/*****************************************************************
*		Datentyp in typlist suchen
******************************************************************/
plcbit iodrv_parser_dptype(unsigned char *pName, unsigned short size)
{

		BOOL	TypFound=0;

		/* -------------------------------------------- */
	 	/* Datenpunkt Eintraege fuer IODRV-Treiber parsen */
		/* -------------------------------------------- */

		/* Parser-Status loeschen */
		State_find_StationTypPoint	= 0;
		State_find_Section			= 0;
		State_find_Data				= 0;

		while (!TypFound && (PaTypList.pParser < (unsigned char*) DOI_typlist.pDatObjMem + DOI_typlist.len) && (State_find_StationTypPoint>=0)) {

			/* Suche nach Stations/Typ/Punkt-Beschreibung */
			State_find_StationTypPoint = find_StationTypPoint (	(unsigned char*) DOI_typlist.pDatObjMem, PaTypList.pParser,
																(unsigned char*) DOI_typlist.pDatObjMem + DOI_typlist.len,
																&PaTypList.pParser, &PaTypList.pParserLine, &PaTypList.pParserErr, &PaTypList.CountLines,
																&PaTypList.pDataArg1, &PaTypList.SizeArg1,
																&PaTypList.pDataArg2, &PaTypList.SizeArg2,
																&PaTypList.SectionType);
			/* keine Daten oder Fehler aufgetreten ? */
			if (State_find_StationTypPoint < 0) {
				break;
			}

			if(PaTypList.SectionType==cCD_TYP) {
				if((PaTypList.SizeArg1==size) && (strncasecmp(PaTypList.pDataArg1, pName, PaTypList.SizeArg1) == 0)) {
					TypFound = 1;

					/* Parserposition zwischenspeichern */
					memcpy(&PaTypListSave,&PaTypList,sizeof(PaTypListSave));

					/* Suchen nach Sektion "IODRV" */
					State_find_Section = find_Section (	(unsigned char*) DOI_typlist.pDatObjMem, PaTypList.pParser,
														(unsigned char*) DOI_typlist.pDatObjMem + DOI_typlist.len,
														&PaTypList.pParser, &PaTypList.pParserLine, &PaTypList.pParserErr, &PaTypList.CountLines,
														&PaTypList.pDataArg1, &PaTypList.SizeArg1,
														&PaTypList.pDataArg2, &PaTypList.SizeArg2,
														KW_IODRV_SECTION);

					/* Section gefunden ? Daten parsen */
					if (State_find_Section == TRUE) {

						/* Pointer auf Anfang der Sektion stellen */
						if (PaTypList.pDataArg2 != NULL) {
							PaTypList.pParser = PaTypList.pDataArg2;
						}
						else {
							continue;
						}

						iodrv_parser_data((unsigned char*) DOI_typlist.pDatObjMem,
										(unsigned char*) DOI_typlist.pDatObjMem + DOI_typlist.len,
										(Parser_typ *) &PaTypList,
										(IODRV_ItemData_typ *) &IODRV_DPData,
										IODRV_SECTION,DP_PART);
					}
					/* Parserposition rückkopieren */
					memcpy(&PaTypList,&PaTypListSave,sizeof(PaTypList));

					/* Suchen nach Sektion "ALL" */
					State_find_Section = find_Section (	(unsigned char*) DOI_typlist.pDatObjMem, PaTypList.pParser,
														(unsigned char*) DOI_typlist.pDatObjMem + DOI_typlist.len,
														&PaTypList.pParser, &PaTypList.pParserLine, &PaTypList.pParserErr, &PaTypList.CountLines,
														&PaTypList.pDataArg1, &PaTypList.SizeArg1,
														&PaTypList.pDataArg2, &PaTypList.SizeArg2,
														KW_ALL_SECTION);

					/* Section gefunden ? Daten parsen */
					if (State_find_Section == TRUE) {

						/* Pointer auf Anfang der Sektion stellen */
						if (PaTypList.pDataArg2 != NULL) {
							PaTypList.pParser = PaTypList.pDataArg2;
						}
						else {
							continue;
						}

						iodrv_parser_data((unsigned char*) DOI_typlist.pDatObjMem,
										(unsigned char*) DOI_typlist.pDatObjMem + DOI_typlist.len,
										(Parser_typ *) &PaTypList,
										(IODRV_ItemData_typ *) &IODRV_DPData,
										ALL_SECTION,DP_PART);
					}
					/* Parserposition rückkopieren */
					memcpy(&PaTypList,&PaTypListSave,sizeof(PaTypList));

				}
			}
		}
	return(TypFound);
}

/*****************************************************************
*		Informationen ueber ein Item ermitteln
******************************************************************/
plcbit iodrv_parser_iteminfo()
{

		BOOL	ItemFound=0;

		/* -------------------------------------------- */
	 	/* Datenpunkt Eintraege fuer IODRV-Treiber parsen */
		/* -------------------------------------------- */

		/* Parser-Status loeschen */
		State_find_StationTypPoint	= 0;
		State_find_Section			= 0;
		State_find_Data				= 0;

		while (!ItemFound && (PaTypList.pParser < (unsigned char*) DOI_typlist.pDatObjMem + DOI_typlist.len)) {

			/* Suche nach Stations/Typ/Punkt-Beschreibung */
			State_find_StationTypPoint = find_StationTypPoint (	(unsigned char*) DOI_typlist.pDatObjMem, PaTypList.pParser,
																(unsigned char*) DOI_typlist.pDatObjMem + DOI_typlist.len,
																&PaTypList.pParser, &PaTypList.pParserLine, &PaTypList.pParserErr, &PaTypList.CountLines,
																&PaTypList.pDataArg1, &PaTypList.SizeArg1,
																&PaTypList.pDataArg2, &PaTypList.SizeArg2,
																&PaTypList.SectionType);
			/* keine Daten oder Fehler aufgetreten ? */
			if (State_find_StationTypPoint < 0) {
				break;
			}

			if(PaTypList.SectionType==cCD_ITEM) {

				/* Parserposition zwischenspeichern */
				memcpy(&PaTypListSave,&PaTypList,sizeof(PaTypListSave));

				/* Suchen nach Sektion "IODRV" */
				State_find_Section = find_Section (	(unsigned char*) DOI_typlist.pDatObjMem, PaTypList.pParser,
													(unsigned char*) DOI_typlist.pDatObjMem + DOI_typlist.len,
													&PaTypList.pParser, &PaTypList.pParserLine, &PaTypList.pParserErr, &PaTypList.CountLines,
													&PaTypList.pDataArg1, &PaTypList.SizeArg1,
													&PaTypList.pDataArg2, &PaTypList.SizeArg2,
													KW_IODRV_SECTION);

				/* keine Daten oder Fehler aufgetreten ? */
				if (State_find_Section < 0) {
					break;
				}

				/* Pointer auf Anfang der Sektion stellen */
				if (PaTypList.pDataArg2 != NULL) {
					PaTypList.pParser = PaTypList.pDataArg2;
				}
				else {
					continue;
				}

				ItemFound	= 1;

				iodrv_parser_data((unsigned char*) DOI_typlist.pDatObjMem,
								(unsigned char*) DOI_typlist.pDatObjMem + DOI_typlist.len,
								(Parser_typ *) &PaTypList,
								(IODRV_ItemData_typ *) &IODRV_ItemData,
								IODRV_SECTION,ITEM_PART);

				/* Parserposition rückkopieren */
				memcpy(&PaTypList,&PaTypListSave,sizeof(PaTypList));

				/* Suchen nach Sektion "ALL" */
				State_find_Section = find_Section (	(unsigned char*) DOI_typlist.pDatObjMem, PaTypList.pParser,
													(unsigned char*) DOI_typlist.pDatObjMem + DOI_typlist.len,
													&PaTypList.pParser, &PaTypList.pParserLine, &PaTypList.pParserErr, &PaTypList.CountLines,
													&PaTypList.pDataArg1, &PaTypList.SizeArg1,
													&PaTypList.pDataArg2, &PaTypList.SizeArg2,
													KW_ALL_SECTION);

				/* keine Daten oder Fehler aufgetreten ? */

				if (State_find_Section>0) {

					/* Pointer auf Anfang der Sektion stellen */
					if (PaTypList.pDataArg2 != NULL) {
						PaTypList.pParser = PaTypList.pDataArg2;
					}
					else {
						continue;
					}

					iodrv_parser_data((unsigned char*) DOI_typlist.pDatObjMem,
									(unsigned char*) DOI_typlist.pDatObjMem + DOI_typlist.len,
									(Parser_typ *) &PaTypList,
									(IODRV_ItemData_typ *) &IODRV_ItemData,
									ALL_SECTION,ITEM_PART);

				}
			}
			else {
				break;
			}

		}

	return(ItemFound);
}

/*****************************************************************
*	Datenbereich einer Sektion parsen
******************************************************************/
void iodrv_parser_data(unsigned char *pSrcStart,unsigned char *pSrcEnd, Parser_typ *pPa, IODRV_ItemData_typ *pData, unsigned char SectionInfo, unsigned char PartInfo) {

	plcbit			dataReady = 0;
	plcbit			dataFound = 0;
	unsigned char	Arg3IsANumber;
	long			Arg3Value;

	do {
		/* Daten der Sektion anfordern */
		State_find_Data = find_Data (	pSrcStart, pPa->pParser, pSrcEnd,
										  &pPa->pParser, &pPa->pParserLine, &pPa->pParserErr, NULL,
										  &pPa->pDataArg1, &pPa->SizeArg1,
										  &pPa->pDataArg2, &pPa->SizeArg2,
										  &pPa->pDataArg3, &pPa->SizeArg3);

		/* Zeilenende erreicht */
		if (State_find_Data == -1) {
			pPa->pParser++;
		}
		/* Daten vorhanden */
		else if (State_find_Data == TRUE) {

			dataFound = 0;

			/* Pruefen, ob Argument 3 einer Zahl entspricht */
			if(pPa->pDataArg3 != NULL && pPa->SizeArg3 != 0) {
				Arg3IsANumber	= IsANumber(pPa->pDataArg3);
				if(Arg3IsANumber==TRUE)	Arg3Value	= brsatoi((UDINT) pPa->pDataArg3);
			}
			else {
				Arg3IsANumber = FALSE;
			}

			/* Schlüsselworte pruefen, die nur im allgemeinen Datenpunktbereich vorkommen */
			if(PartInfo==DP_PART) {
				/* Anlagennummer */
				if (strncasecmp(pPa->pDataArg1, KW_DP_ALL_ANL, pPa->SizeArg1) == 0 && strlen(KW_DP_ALL_ANL) == pPa->SizeArg1 &&
					strncasecmp(pPa->pDataArg2, KW_DP_ALL_ANL_NR, pPa->SizeArg2) == 0 && strlen(KW_DP_ALL_ANL_NR) == pPa->SizeArg2 &&
					Arg3IsANumber  == TRUE) {

						pData->AnlagenNr.value		= Arg3Value;
						pData->AnlagenNr.defined	= 1;
						dataFound					= 1;
				}
				/* Datenpunkt Nummer */
				else if (strncasecmp(pPa->pDataArg1, KW_DP_ALL_DP, pPa->SizeArg1) == 0 && strlen(KW_DP_ALL_DP) == pPa->SizeArg1 &&
						strncasecmp(pPa->pDataArg2, KW_DP_ALL_DP_NR, pPa->SizeArg2) == 0 && strlen(KW_DP_ALL_DP_NR) == pPa->SizeArg2 &&
						Arg3IsANumber == TRUE) {
						/* Nummer der Anlage */
						pData->DPNr.value			= Arg3Value;
						pData->DPNr.defined			= 1;
						dataFound					= 1;
				}
				/* Datentyp */
				else if (strncasecmp(pPa->pDataArg1, KW_DP_ALL_TYP, pPa->SizeArg1) == 0 && strlen(KW_DP_ALL_TYP) == pPa->SizeArg1 &&
						pPa->SizeArg2==0 &&
						pPa->pDataArg3 != NULL && pPa->SizeArg3 != 0) {

						pData->Typ.name				= pPa->pDataArg3;
						pData->Typ.size				= pPa->SizeArg3;
						pData->Typ.defined			= 1;
						dataFound					= 1;
				}
				/* Datentyp Item */
				else if (strncasecmp(pPa->pDataArg1, KW_DP_ALL_ITEM, pPa->SizeArg1) == 0 && strlen(KW_DP_ALL_ITEM) == pPa->SizeArg1 &&
						strncasecmp(pPa->pDataArg2, KW_DP_ALL_ITEM_TYP, pPa->SizeArg2) == 0 && strlen(KW_DP_ALL_ITEM_TYP) == pPa->SizeArg2 &&
						pPa->pDataArg3 != NULL && pPa->SizeArg3 != 0) {

						pData->ItemTyp.name			= pPa->pDataArg3;
						pData->ItemTyp.size			= pPa->SizeArg3;
						pData->ItemTyp.defined		= 1;
						dataFound					= 1;
				}
				/* Item Nummer */
				else if (strncasecmp(pPa->pDataArg1, KW_DP_ALL_ITEM, pPa->SizeArg1) == 0 && strlen(KW_DP_ALL_ITEM) == pPa->SizeArg1 &&
						strncasecmp(pPa->pDataArg2, KW_DP_ALL_ITEM_NR, pPa->SizeArg2) == 0 && strlen(KW_DP_ALL_ITEM_NR) == pPa->SizeArg2 &&
						Arg3IsANumber == TRUE) {

						pData->ItemNr.value			= Arg3Value;
						pData->ItemNr.defined		= 1;
						dataFound					= 1;
				}
				/* Item Name */
				else if (strncasecmp(pPa->pDataArg1, KW_DP_ALL_ITEM, pPa->SizeArg1) == 0 && strlen(KW_DP_ALL_ITEM) == pPa->SizeArg1 &&
						strncasecmp(pPa->pDataArg2, KW_DP_ALL_ITEM_NAME, pPa->SizeArg2) == 0 && strlen(KW_DP_ALL_ITEM_NAME) == pPa->SizeArg2 &&
						pPa->pDataArg3 != NULL && pPa->SizeArg3 != 0) {

						pData->ItemName.name		= pPa->pDataArg3;
						pData->ItemName.size		= pPa->SizeArg3;
						pData->ItemName.defined		= 1;
						dataFound					= 1;
				}
				/* invers */
				else if (strncasecmp(pPa->pDataArg1, KW_ITEM_IODRV_INV, pPa->SizeArg1) == 0 && strlen(KW_ITEM_IODRV_INV) == pPa->SizeArg1 &&
						pPa->SizeArg2==0 &&
						Arg3IsANumber  == TRUE) {

						/* invers */
						pData->Invers.value			= Arg3Value;
						pData->Invers.defined		= 1;
						dataFound					= 1;
				}
				/* Quitt */
				else if (strncasecmp(pPa->pDataArg1, KW_ITEM_IODRV_QUITT, pPa->SizeArg1) == 0 && strlen(KW_ITEM_IODRV_QUITT) == pPa->SizeArg1 &&
						pPa->SizeArg2==0 &&
						Arg3IsANumber == TRUE) {

						pData->Quitt.value			= Arg3Value;
						pData->Quitt.defined		= 1;
						if(Arg3Value)	{
							/* bei Quittierpflichtigem Item: Attr = ReadWrite */
							pData->Dir.value			= cKW_READWRITE;
							pData->Dir.defined			= 1;
						}
						dataFound					= 1;
				}
				/* Dir (als Zahl 0/1/2)*/
				else if (strncasecmp(pPa->pDataArg1, KW_ITEM_IODRV_DIR, pPa->SizeArg1) == 0 && strlen(KW_ITEM_IODRV_DIR) == pPa->SizeArg1 &&
						pPa->SizeArg2==0 &&
						Arg3IsANumber == TRUE) {

						pData->Dir.value			= Arg3Value;
						pData->Dir.defined			= 1;
						dataFound					= 1;
				}
				/* Dir (als Text R/W/RW)*/
				else if (strncasecmp(pPa->pDataArg1, KW_ITEM_IODRV_DIR, pPa->SizeArg1) == 0 && strlen(KW_ITEM_IODRV_DIR) == pPa->SizeArg1 &&
						pPa->SizeArg2==0 &&
						pPa->pDataArg3 != NULL && pPa->SizeArg3 != 0) {

						if(!strncasecmp(pPa->pDataArg3,KW_ITEM_IODRV_DIR_R,pPa->SizeArg3))	{
							pData->Dir.value			= cKW_READ;
							pData->Dir.defined			= 1;
							dataFound					= 1;
						}
						else if(!strncasecmp(pPa->pDataArg3,KW_ITEM_IODRV_DIR_W,pPa->SizeArg3))	{
							pData->Dir.value			= cKW_WRITE;
							pData->Dir.defined			= 1;
							dataFound					= 1;
						}
						else if(!strncasecmp(pPa->pDataArg3,KW_ITEM_IODRV_DIR_RW,pPa->SizeArg3))	{
							pData->Dir.value			= cKW_READWRITE;
							pData->Dir.defined			= 1;
							dataFound					= 1;
						}
				}
				/* Datentyp Nummer */
				else if (strncasecmp(pPa->pDataArg1, KW_DPTYP_ALL_TYP, pPa->SizeArg1) == 0 && strlen(KW_DPTYP_ALL_TYP) == pPa->SizeArg1 &&
						strncasecmp(pPa->pDataArg2, KW_DPTYP_ALL_TYP_NR, pPa->SizeArg2) == 0 && strlen(KW_DPTYP_ALL_TYP_NR) == pPa->SizeArg2 &&
						Arg3IsANumber == TRUE) {

						pData->DPTypNr.value		= Arg3Value;
						pData->DPTypNr.defined		= 1;
						dataFound					= 1;
				}
			}

			if(PartInfo==ITEM_PART) {
				/* Datentyp Item */
				if (strncasecmp(pPa->pDataArg1, KW_ITEM_ALL_ITEM_TYP, pPa->SizeArg1) == 0 && strlen(KW_ITEM_ALL_ITEM_TYP) == pPa->SizeArg1 &&
						pPa->SizeArg2==0 &&
						pPa->pDataArg3 != NULL && pPa->SizeArg3 != 0) {

						pData->ItemTyp.name			= pPa->pDataArg3;
						pData->ItemTyp.size			= pPa->SizeArg3;
						pData->ItemTyp.defined		= 1;
						dataFound					= 1;
				}
				/* Item Nummer */
				else if (strncasecmp(pPa->pDataArg1, KW_ITEM_ALL_ITEM, pPa->SizeArg1) == 0 && strlen(KW_ITEM_ALL_ITEM) == pPa->SizeArg1 &&
						strncasecmp(pPa->pDataArg2, KW_ITEM_ALL_ITEM_NR, pPa->SizeArg2) == 0 && strlen(KW_ITEM_ALL_ITEM_NR) == pPa->SizeArg2 &&
						Arg3IsANumber == TRUE) {

						pData->ItemNr.value			= Arg3Value;
						pData->ItemNr.defined		= 1;
						dataFound					= 1;
				}
				/* Item Name */
				else if (strncasecmp(pPa->pDataArg1, KW_DP_ALL_ITEM, pPa->SizeArg1) == 0 && strlen(KW_DP_ALL_ITEM) == pPa->SizeArg1 &&
						strncasecmp(pPa->pDataArg2, KW_DP_ALL_ITEM_NAME, pPa->SizeArg2) == 0 && strlen(KW_DP_ALL_ITEM_NAME) == pPa->SizeArg2 &&
						pPa->pDataArg3 != NULL && pPa->SizeArg3 != 0) {

						pData->ItemName.name		= pPa->pDataArg3;
						pData->ItemName.size		= pPa->SizeArg3;
						pData->ItemName.defined		= 1;
						dataFound					= 1;
				}
			}

			if(((PartInfo==ITEM_PART) || (PartInfo==DP_PART)) && (!dataFound)) {
				/* invers */
				if (strncasecmp(pPa->pDataArg1, KW_ITEM_IODRV_INV, pPa->SizeArg1) == 0 && strlen(KW_ITEM_IODRV_INV) == pPa->SizeArg1 &&
						pPa->SizeArg2==0 &&
						Arg3IsANumber  == TRUE) {

						/* invers */
						pData->Invers.value			= Arg3Value;
						pData->Invers.defined		= 1;
						dataFound					= 1;
				}
				/* Quitt */
				else if (strncasecmp(pPa->pDataArg1, KW_ITEM_IODRV_QUITT, pPa->SizeArg1) == 0 && strlen(KW_ITEM_IODRV_QUITT) == pPa->SizeArg1 &&
						pPa->SizeArg2==0 &&
						Arg3IsANumber == TRUE) {

						pData->Quitt.value			= Arg3Value;
						pData->Quitt.defined		= 1;
						if(Arg3Value)	{
							/* bei Quittierpflichtigem Item: Attr = ReadWrite */
							pData->Dir.value			= cKW_READWRITE;
							pData->Dir.defined			= 1;
						}
						dataFound					= 1;
				}
				/* Dir (als Zahl 0/1/2)*/
				else if (strncasecmp(pPa->pDataArg1, KW_ITEM_IODRV_DIR, pPa->SizeArg1) == 0 && strlen(KW_ITEM_IODRV_DIR) == pPa->SizeArg1 &&
						pPa->SizeArg2==0 &&
						Arg3IsANumber == TRUE) {

						pData->Dir.value			= Arg3Value;
						pData->Dir.defined			= 1;
						dataFound					= 1;
				}
				/* Dir (als Text R/W/RW)*/
				else if (strncasecmp(pPa->pDataArg1, KW_ITEM_IODRV_DIR, pPa->SizeArg1) == 0 && strlen(KW_ITEM_IODRV_DIR) == pPa->SizeArg1 &&
						pPa->SizeArg2==0 &&
						pPa->pDataArg3 != NULL && pPa->SizeArg3 != 0) {

						if(!strncasecmp(pPa->pDataArg3,KW_ITEM_IODRV_DIR_R,pPa->SizeArg3))	{
							pData->Dir.value			= cKW_READ;
							pData->Dir.defined			= 1;
							dataFound					= 1;
						}
						else if(!strncasecmp(pPa->pDataArg3,KW_ITEM_IODRV_DIR_W,pPa->SizeArg3))	{
							pData->Dir.value			= cKW_WRITE;
							pData->Dir.defined			= 1;
							dataFound					= 1;
						}
						else if(!strncasecmp(pPa->pDataArg3,KW_ITEM_IODRV_DIR_RW,pPa->SizeArg3))	{
							pData->Dir.value			= cKW_READWRITE;
							pData->Dir.defined			= 1;
							dataFound					= 1;
						}
				}
			}

			/* Unbekannter Eintrag */
			if((!dataFound) && (SectionInfo==IODRV_SECTION)) {
				iodrv_parser_warn(PARS_ERR_UNKNOWN_ITEM_ENTRY,"Unbekannter Eintrag im Item-Bereich:", pPa->pParserLine, " / Zeile =", (long) pPa->CountLines, 0, 0, 0, 0);
			}
		}

		/* Endebedinung der Schleife: Keine Daten mehr vorhanden, oder Ende des Datenmodules erreicht */
		if((State_find_Data!=TRUE) && (State_find_Data!=-1))	dataReady = 1;
		if(pPa->pParser >= pSrcEnd)	dataReady = 1;
	} while (!dataReady);
}

/*****************************************************************
*	Pruefen, ob alle Angaben eines Datenpunktes vorhanden sind
******************************************************************/
plcbit iodrv_parser_dpinfo_ok(IODRV_ItemData_typ *pData)
{
	plcbit ok;

	ok = 1;
	if(!pData->AnlagenNr.defined) {
		iodrv_parser_warn(PARS_ERR_ANLNR_NOT_DEFINED,"DP Anlage.Nr fehlt. DPTyp: ", pData->Typ.name ,"DPNr.", pData->DPNr.value, 0, 0, 0, 0);
		ok = 0;
	}
	if(!pData->DPNr.defined) {
		iodrv_parser_warn(PARS_ERR_DPNR_NOT_DEFINED,"DP DP.Nr fehlt. DPTyp: ", pData->Typ.name , 0, 0, 0, 0, 0, 0);
		ok = 0;
	}
	if(!pData->Typ.defined) {
		iodrv_parser_warn(PARS_ERR_TYP_NOT_DEFINED,"DP Typbezeichnung fehlt. DPTyp: ", 0, "DPNr.", pData->DPNr.value, 0, 0, 0, 0);
		ok = 0;
	}

	return(ok);
}

/*****************************************************************
*	Pruefen, ob alle Angaben eines Items vorhanden sind
******************************************************************/
plcbit iodrv_parser_iteminfo_ok(IODRV_ItemData_typ *pData)
{

	plcbit	ok;

	ok = 1;
	/* Datentyp Nummer definiert ? */
	if(!pData->DPTypNr.defined) {
		iodrv_parser_warn(PARS_ERR_DPTYP_NR_NOT_DEFINED,"Typ.Nr fehlt. DPTyp: ", pData->Typ.name , "DPNr.", pData->DPNr.value, 0, 0, 0, 0);
		ok = 0;
	}

	/* Item Nummer definiert ? */
	if(!pData->ItemNr.defined) {
		iodrv_parser_warn(PARS_ERR_ITEM_NR_NOT_DEFINED,"Item.Nr fehlt. DPTyp: ", pData->Typ.name , "DPNr.", pData->DPNr.value, 0, 0, 0, 0);
		ok = 0;
	}

	/* Item Typ definiert ? */
	if(!pData->ItemTyp.defined) {
		iodrv_parser_warn(PARS_ERR_ITEM_TYP_NOT_DEFINED,"ITEM Datentyp fehlt. DPTyp: ", pData->Typ.name , "DPNr.", pData->DPNr.value, "Item-Nr.", pData->ItemNr.value, 0, 0);
		ok = 0;
	}
	else {
		pData->ItemTypNr.defined = 0;
		/* Item Datentyp gültig ? */
		if(strncasecmp(pData->ItemTyp.name, BOOL_TYP, pData->ItemTyp.size) == 0 && strlen(BOOL_TYP) == pData->ItemTyp.size) {
			pData->ItemTypNr.defined	= 1;
			pData->ItemTypNr.value		= BOOL_IDX;
		}
		if(strncasecmp(pData->ItemTyp.name, USINT_TYP, pData->ItemTyp.size) == 0 && strlen(USINT_TYP) == pData->ItemTyp.size) {
			pData->ItemTypNr.defined	= 1;
			pData->ItemTypNr.value		= USINT_IDX;
		}
		if(strncasecmp(pData->ItemTyp.name, SINT_TYP, pData->ItemTyp.size) == 0 && strlen(SINT_TYP) == pData->ItemTyp.size) {
			pData->ItemTypNr.defined	= 1;
			pData->ItemTypNr.value		= SINT_IDX;
		}
		if(strncasecmp(pData->ItemTyp.name, UINT_TYP, pData->ItemTyp.size) == 0 && strlen(UINT_TYP) == pData->ItemTyp.size) {
			pData->ItemTypNr.defined	= 1;
			pData->ItemTypNr.value		= UINT_IDX;
		}
		if(strncasecmp(pData->ItemTyp.name, INT_TYP, pData->ItemTyp.size) == 0 && strlen(INT_TYP) == pData->ItemTyp.size) {
			pData->ItemTypNr.defined	= 1;
			pData->ItemTypNr.value		= INT_IDX;
		}
		if(strncasecmp(pData->ItemTyp.name, UDINT_TYP, pData->ItemTyp.size) == 0 && strlen(UDINT_TYP) == pData->ItemTyp.size) {
			pData->ItemTypNr.defined	= 1;
			pData->ItemTypNr.value		= UDINT_IDX;
		}
		if(strncasecmp(pData->ItemTyp.name, DINT_TYP, pData->ItemTyp.size) == 0 && strlen(DINT_TYP) == pData->ItemTyp.size) {
			pData->ItemTypNr.defined	= 1;
			pData->ItemTypNr.value		= DINT_IDX;
		}
		if(!pData->ItemTypNr.defined) {
			iodrv_parser_warn(PARS_ERR_ITEM_TYP_UNKNOWN,"ITEM Datentyp unbekannt. DPTyp: ", pData->Typ.name , "DPNr.", pData->DPNr.value, "Item-Nr.", pData->ItemNr.value, 0, 0);
			ok = 0;
		}
	}
	/* Item Name definiert ? */
	if(!pData->ItemName.defined) {
		iodrv_parser_warn(PARS_ERR_ITEM_NAME_NOT_DEFINED,"ITEM Itemname fehlt. DPTyp: ", pData->Typ.name , "DPNr.", pData->DPNr.value, "Item-Nr.", pData->ItemNr.value, 0, 0);
		ok = 0;
	}

	/* Invers definiert ? */
	if(!pData->Invers.defined) {
		iodrv_parser_warn(PARS_ERR_IODRV_INV_NOT_DEFINED,"ITEM Invers fehlt. DPTyp: ", pData->Typ.name , "DPNr.", pData->DPNr.value, "Item-Nr.", pData->ItemNr.value, 0, 0);
		ok = 0;
	}

	/* Quitt definiert ? */
	if(!pData->Quitt.defined) {
		iodrv_parser_warn(PARS_ERR_IODRV_QUITT_NOT_DEFINED,"ITEM Quitt fehlt. DPTyp: ", pData->Typ.name , "DPNr.", pData->DPNr.value, "Item-Nr.", pData->ItemNr.value, 0, 0);
		ok = 0;
	}

	return(ok);
}

/***************************************************************************
*		Zeiger auf Startadresse Datenmodul stellen, Zeilenzaehler loeschen
****************************************************************************/
void copyItemData(IODRV_ItemData_typ *pItemDest, IODRV_ItemData_typ *pItemSrc)
{
	if(pItemSrc->AnlagenNr.defined)		memcpy(&pItemDest->AnlagenNr,	&pItemSrc->AnlagenNr,	sizeof(pItemDest->AnlagenNr));
	if(pItemSrc->DPNr.defined)			memcpy(&pItemDest->DPNr,		&pItemSrc->DPNr,		sizeof(pItemDest->DPNr));
	if(pItemSrc->DPTypNr.defined)		memcpy(&pItemDest->DPTypNr,		&pItemSrc->DPTypNr,		sizeof(pItemDest->DPTypNr));
	if(pItemSrc->DPName.defined)		memcpy(&pItemDest->DPName,		&pItemSrc->DPName,		sizeof(pItemDest->DPName));
	if(pItemSrc->Typ.defined)			memcpy(&pItemDest->Typ,			&pItemSrc->Typ,			sizeof(pItemDest->Typ));
	if(pItemSrc->ItemNr.defined)		memcpy(&pItemDest->ItemNr,		&pItemSrc->ItemNr,		sizeof(pItemDest->ItemNr));
	if(pItemSrc->ItemTyp.defined)		memcpy(&pItemDest->ItemTyp,		&pItemSrc->ItemTyp,		sizeof(pItemDest->ItemTyp));
	if(pItemSrc->ItemName.defined)		memcpy(&pItemDest->ItemName,	&pItemSrc->ItemName,	sizeof(pItemDest->ItemName));
	if(pItemSrc->Invers.defined)		memcpy(&pItemDest->Invers,		&pItemSrc->Invers,		sizeof(pItemDest->Invers));
	if(pItemSrc->Quitt.defined)			memcpy(&pItemDest->Quitt,		&pItemSrc->Quitt,		sizeof(pItemDest->Quitt));
	if(pItemSrc->Dir.defined)			memcpy(&pItemDest->Dir,			&pItemSrc->Dir,			sizeof(pItemDest->Dir));
}

/***************************************************************************
*		Zeiger auf Startadresse Datenmodul stellen, Zeilenzaehler loeschen
****************************************************************************/
void iodrv_parser_dplist_clear()
{

	/* Datenmodul von Anfang an Parsen .. */
	PaDPList.pParser		= (unsigned char*) DOI_dplist.pDatObjMem;
	PaDPList.CountLines		= 0;
}

/***************************************************************************
*		Zeiger auf Startadresse Datenmodul stellen, Zeilenzaehler loeschen
****************************************************************************/
void iodrv_parser_typlist_clear()
{

	/* Datenmodul von Anfang an Parsen ... */
	PaTypList.pParser		= (unsigned char*) DOI_typlist.pDatObjMem;
	PaTypList.CountLines	= 0;
}
/**********************************************************
*		Fehlermeldung in Log-Buch eintragen
**********************************************************/
void iodrv_parser_err(unsigned short errorNr, unsigned char *pTxtInfo, unsigned char *pTxt0, unsigned char *pTxt1, long info1, unsigned char *pTxt2, long info2, unsigned char *pTxt3, long info3)
{
	unsigned char ANr[20];
	unsigned long ErrorInfo=0;

	memset(MsgTxt,0,sizeof(MsgTxt));
	if(IODRV_ParserInfo.ErrorMsg) {
		IODRV_ParserInfo.error = errorNr;
		strcpy(MsgTxt," ");
		if(pTxtInfo>0) {
			strcat(MsgTxt,pTxtInfo);
			strcat(MsgTxt," ");
		}
		if(pTxt0>0) {
			strcat(MsgTxt,pTxt0);
			strcat(MsgTxt," ");
		}
		if(pTxt1>0) {
			strcat(MsgTxt,pTxt1);
			strcat(MsgTxt," ");
			brsitoa(info1, (UDINT) &ANr);
			strcat(MsgTxt,ANr);
			strcat(MsgTxt," ");
		}
		if(pTxt2>0) {
			strcat(MsgTxt,pTxt2);
			strcat(MsgTxt," ");
			brsitoa(info2, (UDINT) &ANr);
			strcat(MsgTxt,ANr);
			strcat(MsgTxt," ");
		}
		if(pTxt3>0) {
			strcat(MsgTxt,pTxt3);
			strcat(MsgTxt," ");
			brsitoa(info3, (UDINT) &ANr);
			strcat(MsgTxt,ANr);
			strcat(MsgTxt," ");
		}
		if(IODRV_ParserInfo.NrOfLogEntrys>MAX_ERROR_MSG_LOG) {
			ErrStatistics("iodrv", ERR, errorNr, ErrorInfo, ERR_MSG_PRE_STRG, MsgTxt);
		}
		else {
			ErrStatistics("iodrv", ERRLOG, errorNr, ErrorInfo, ERR_MSG_PRE_STRG, MsgTxt);
		}
		IODRV_ParserInfo.NrOfLogEntrys++;
	}
}

/**********************************************************
*		Warnungsmeldung in Log-Buch eintragen
**********************************************************/
void iodrv_parser_warn(unsigned short warnNr, unsigned char *pTxtInfo, unsigned char *pTxt0, unsigned char *pTxt1, long info1, unsigned char *pTxt2, long info2, unsigned char *pTxt3, long info3)
{
	unsigned char ANr[20];
	unsigned long ErrorInfo=0;

	memset(MsgTxt,0,sizeof(MsgTxt));
	if(IODRV_ParserInfo.ErrorMsg) {
		IODRV_ParserInfo.warning = warnNr;
		strcpy(MsgTxt," ");
		if(pTxtInfo>0) {
			strcat(MsgTxt,pTxtInfo);
			strcat(MsgTxt," ");
		}
		if(pTxt0>0) {
			strcat(MsgTxt,pTxt0);
			strcat(MsgTxt," ");
		}
		if(pTxt1>0) {
			strcat(MsgTxt,pTxt1);
			strcat(MsgTxt," ");
			brsitoa(info1, (UDINT) &ANr);
			strcat(MsgTxt,ANr);
			strcat(MsgTxt," ");
		}
		if(pTxt2>0) {
			strcat(MsgTxt,pTxt2);
			strcat(MsgTxt," ");
			brsitoa(info2, (UDINT) &ANr);
			strcat(MsgTxt,ANr);
			strcat(MsgTxt," ");
		}
		if(pTxt3>0) {
			strcat(MsgTxt,pTxt3);
			strcat(MsgTxt," ");
			brsitoa(info3, (UDINT) &ANr);
			strcat(MsgTxt,ANr);
			strcat(MsgTxt," ");
		}
		if(IODRV_ParserInfo.NrOfLogEntrys>MAX_ERROR_MSG_LOG) {
			ErrStatistics("iodrv", ERR, warnNr, ErrorInfo, ERR_MSG_PRE_STRG, MsgTxt);
		}
		else {
			ErrStatistics("iodrv", ERRLOG, warnNr, ErrorInfo, ERR_MSG_PRE_STRG, MsgTxt);
		}
		IODRV_ParserInfo.NrOfLogEntrys++;
	}
}

/**********************************************************
*		Speicherdiagnose
**********************************************************/
void iodrv_mem_diagnose()
{
	IODRV_DP_Info_typ *pDPInfo;
	unsigned short	n,i;
	plcbit			found;

	for(i=0;i<ITEM_DIAGNOSE_SIZE;i++) {
		if(IODRV_ItemDiagnose[i].showData) {
			IODRV_ItemDiagnose[i].showData	= 0;
			IODRV_ItemDiagnose[i].DataValid	= 0;

			found = 0;
			pDPInfo = (IODRV_DP_Info_typ *) (IODRV_ParserInfo.memAdr);
			for(n = 0; n < IODRV_ParserInfo.NrOfItems; n++, pDPInfo++) {
				if(IODRV_ItemDiagnose[i].AnlagenNr 	!= pDPInfo->AnlagenNr)	continue;
				if(IODRV_ItemDiagnose[i].DPTypNr 	!= pDPInfo->DPTypNr)	continue;
				if(IODRV_ItemDiagnose[i].DPNr 		!= pDPInfo->DPNr)	continue;
				if(IODRV_ItemDiagnose[i].ItemNr 	!= pDPInfo->ItemNr)		continue;
				found = 1;
				IODRV_ItemDiagnose[i].ItemIdx = n;
				break;
			}

			if(found) {
				IODRV_ItemDiagnose[i].pItemData		 = (IODRV_DP_Info_typ *)  (IODRV_ParserInfo.memAdr);
				IODRV_ItemDiagnose[i].pItemData		+= IODRV_ItemDiagnose[i].ItemIdx;
				IODRV_ItemDiagnose[i].DataValid	 = 1;
				if(i==0) {
					pItemData0Diagnose = IODRV_ItemDiagnose[i].pItemData;
				}
				else {
					pItemData1Diagnose = IODRV_ItemDiagnose[i].pItemData;
				}
			}
		}
	}
}

/***********************************************************************/
/* Tcp-Funktionen                                                      */
/***********************************************************************/

unsigned char IsANumber(unsigned char *pData) {

	unsigned char	flag;
	unsigned short	i;

#define	cMAX_CHARACTERS	16

	flag = FALSE;
	if (pData != NULL) {
		for (i=0; i<cMAX_CHARACTERS; i++) {
			if (pData[i] == 0) {
				break;
			}
			else if (pData[i] == ' ' && flag == TRUE) {
				break;
			}
			else if (pData[i]>='0' && pData[i]<='9') {
				flag = TRUE;
			}
			else {
				break;
			}
		}
		if (i == cMAX_CHARACTERS) {
			flag = FALSE;
		}
	}
	return flag;
}

/*** eof *****************************************************************************/
```

#### iodrv_sub.c
```c
#ifdef _DEFAULT_INCLUDES
	#include <AsDefault.h>
#endif
/******************************************************************************
*    COPYRIGHT    BERNECKER + RAINER Industrie-Elektronik Ges.m.b.H           *
*******************************************************************************
*  Projekt:  I/O-Treiber
*  Teil:     Unterprogramme
*  Datei:    iodrv_sub.c
*  Typ:      GNU-C (32 Bit)
*------------------------------------------------------------------------------
*  Revision: 01.00
*  Datum:    05-04-2006
*  Autor:    WAI
*------------------------------------------------------------------------------
*  Funktion:
*------------------------------------------------------------------------------
*  Rev.  | Datum    | Name | Kommentar
*  ------+----------+------+---------------------------------------------------
*  01.00 | 05-04-06 | WAI  | Datei-Erstellung
*        |          |      |
******************************************************************************/
#include <bur/plctypes.h>
#include <sys_lib.h>		/* SYS_LIB */
#include <fileio.h>
#include "iodrv.h"
#include "dbserv.h"
#include "platform.h"
/****************************************************************************/
/*		BR-Server ID besorgen												*/
/****************************************************************************/
void get_idBrServer() {

	if (myidBrServer == 0) {
		idstat = GetIdBrServer((void*)&myidBrServer,&brstate);
	}
}
```

#### iodrv.h
```c
/******************************************************************************
*    COPYRIGHT    BERNECKER + RAINER Industrie-Elektronik Ges.m.b.H           *
*******************************************************************************
*  Projekt:  I/O-Treiber
*  Teil:     Headerfile
*  Datei:    iodrv.h
*  Typ:      GNU-C (32 Bit)
*------------------------------------------------------------------------------
*  Revision: 01.00
*  Datum:    05-04-2006
*  Autor:    WAI
*------------------------------------------------------------------------------
*  Funktion:
*------------------------------------------------------------------------------
*  Rev.  | Datum    | Name | Kommentar
*  ------+----------+------+---------------------------------------------------
*  01.00 | 05-04-06 | WAI  | Datei-Erstellung
*        |          |      |
******************************************************************************/
#include <bur/plctypes.h>
#include <dvframe.h>
#include <sys_lib.h>
#include <dataobj.h>
#include <brsystem.h>
#include "bksys.h"

/***********************************************************************/
/* Konstantendefinition                                                */
/***********************************************************************/

/* -------------------------------------------*/
/* Grenzwert fuer Linien und Geraete pro Linie */
/* -------------------------------------------*/

#define MAX_LINES							1				/* Maximal moegliche Anzahl Linien */
#define DEVICES_PRO_LINE					128				/* Anzahl moeglicher Geraete pro Linie */

/* --------------------------------------------*/
/* Allgemeine Konstanten                       */
/* --------------------------------------------*/

#define FALSE			0
#define TRUE			1

#define ACK				254
#define NAK				255

#define WRITE			0
#define READ			1

#define INIT_KE			1
#define INIT_KE_LAEUFT	2
#define ZEIT_SYNC		3
#define INIT_GI			4
#define INIT_GI_START   5
#define INIT_GI_LAEUFT	6
#define CLASS_1_REQ		7
#define CLASS_2_REQ		8
#define READY			99

#define TYPE_CONNECTION_ERROR	255		/* Typ für Datenpunkt : Verbindungsfehler */
#define INFO_CONNECTION_ERROR	255		/* Info für Datenpunkt: Verbindungsfehler */

/* -------------------------------------------------------------*/
/* Kennzeichnung für Einzelschritte der Störschriebübermittlung */
/* -------------------------------------------------------------*/

#define NO_FUNCTION							0
#define SELECTION_OF_FAULT	 				1
#define REQ_DISTURBANCE_TRANSMISSION		2
#define REQ_FOR_TAGS						3
#define REQ_FOR_A_CHANNEL					4
#define ACK_FOR_TAGS						5
#define ACK_FOR_A_CHANNEL					6
#define ACK_FOR_DISTURBANCE_DATA			7
#define REQ_FOR_LIST_OF_FAULTS				8
#define ABORT_DISTURBANCE_TRANSMISSION		9
#define ABORT_CHANNEL_TRANSMISSION			10

/* -------------------------------------------------------------------------*/
/* Kennung fuer Stoerschriebbuffer und Stoerschriebinformation des Geraetes */
/* -------------------------------------------------------------------------*/

#define NODATA								0
#define WRITE_BUFFER						1
#define DATA_READY							2
#define WAIT_FOR_QUIT						3
#define DELETE_DATA							4
#define SEND_DELETE_TELEGRAM				5
#define CLEAR_DATA_AGAIN					6

/***********************************************************************/
/* Datentypdeklaration                                                 */
/***********************************************************************/

/* ----------------------------------------*/
/* Konfigurationsvariable des IODRV-Treibers */
/* ----------------------------------------*/
typedef struct
{
	unsigned long			TimeOut;					/* Timeout bei Telegrammempfang (in ms) */
	unsigned short			RetryAnz;					/* Anzahl Telegrammwiederholungen bei bestehender Verbindung */
	unsigned short			ConnAnz;					/* Anzahl Telegrammwiederholung bei neu aufzubauender Verbindung */
	unsigned long			WaitIntv;					/* Wartezeit für erneuten Verbindungsaufbau (in ms) */
	unsigned long			TimeTS;						/* Intervallzeit fuer Uhrzeitsynchronisation (in ms) */
	unsigned short			EnableComReset;				/* Freigabe fuer das Schliessen und Wieder-Oeffnen der Schnittstelle bei Schreibfehlern */
	unsigned long			TimeClass2Poll;				/* Abtastzeit Class 2 Telegramme (Analogwerte) (in ms) */
	unsigned long			TimeClass2PollFast;			/* Abtastzeit Class 2 Telegramme (Analogwerte) während Übertragung von Störschrieben (in ms) */
	unsigned short			DistDataEnable;				/* Freigabe fuer Stoerschriebuebertragung */
	unsigned long			DistDataTimeoutMax;			/* Timeout fuer den Telegrammempfang bei Stoerschriebuebertragung in (ms) */
	unsigned long			DisturbanceDelay;			/* Zeit die ein Lesen von Stoerschrieben der gleichen Station verzoegert wird in (ms) */
	unsigned short			CommandEnable;				/* Freigabe fuer Kommandouebertragung */
	unsigned long			CommandTimeoutMax;			/* Timeout fuer die Uebertragung von Kommandos in (ms) */
} IODRV_Config_typ;

/* Verwaltung der Unterstationen */
/* Struktur eines Datenpunkt Items im Speicher */
typedef struct {
	UINT	AnlagenNr;						/* Anlagennummer eines Geräts */
	UINT	DPTypNr;						/* Datentypnummer */
	UINT	DPNr;							/* Datenpunktnummer */
	UINT	ItemNr;							/* Item Nummer */
	USINT	ItemTypNr;						/* Datentypnummer des Items */
	USINT	*DPName;						/* Datenpunktname */
	UINT	DPNameLen;						/* Länge des DP-Namens */
	USINT	*ItemName;						/* Item Name */
	UINT	ItemNameLen;					/* Länge des Item-Namens */

	USINT	Invers;							/* DP invertieren */
	USINT	Quitt;							/* DP quittierpflichtig */
	USINT	Dir;							/* Schreib-/Leseattribut */

	STRING	PVName[64];						/* Name der PV */
	UDINT	PVAdrs;							/* Adresse der PV */
	UDINT	PVDataLen;						/* Länge der PV */
	DINT	ValueIO;						/* Wert,der vom Geraet empfangen wurde */
	DINT	ValueServer;					/* Wert, der an den Server uebergeben wurde */

	USINT	AccessCounter;					/* Zaehle fuer Zugriffe auf das Item */
	USINT	ErrorInfo;						/* Fehlerinformation */

} IODRV_DP_Info_typ;
/*---------------------------------------------*/
/* Datenmodulstrukturen 		               */
/*---------------------------------------------*/

/*-----------------------------------------------*/
/* Strukturen fuer die Verwaltung eines Geraetes */
/*-----------------------------------------------*/

typedef struct {
	USINT	Nummer;
	USINT	Adresse;
	USINT	Aktiv;
	USINT	TimeSynch;
	UINT	AnlagenNr;
	UINT	Frei;
} DeviceType;

typedef union
{
	BOOL 	b;
	SINT 	i1;
	USINT	ui1;
	INT		i2;
	UINT	ui2;
	DINT	i4;
	UDINT	ui4;
	float r4;
} PAR_TYPE;

/**********************************************************
*						Prototypen
**********************************************************/
/*
USINT save_analogwert(	DMInfoType *pDMInfo,  IODRV_DeviceActivType *pDeviceActiv,
						USINT FunctionType, USINT InformationNumber, USINT AnzahlMesswerte,
						USINT *AdresseMesswerte, USINT set_event);

void save_analogwert_error(	DMInfoType *pDMInfo, IODRV_DeviceActivType *pDeviceActiv,
						USINT FunctionType,USINT InformationNumber, USINT set_event);

USINT save_digitalwert( DMInfoType *pDMInfo, IODRV_DeviceActivType *pDeviceActiv,
						USINT FunctionType,USINT InformationNumber, USINT Messwert,
						RTCtime_typ *TimeBuf, USINT set_event);

USINT save_kopplungsstoerung( DMInfoType *pDMInfo, IODRV_DeviceActivType *pDeviceActiv, USINT Messwert, RTCtime_typ *TimeBuf, USINT set_event);

*/
void debug_initialize(void);

void get_idBrServer();

/**********************************************************
*				Globale Variablen Declaration
**********************************************************/

/**********************************************************
*				Lokale Variablen Declaration
**********************************************************/

_LOCAL	UDINT							myidBrServer;
_LOCAL_RETAIN	UINT							statePV_xgetadr	;
_LOCAL  UINT							StatusSetValueItem;

_LOCAL	RTInfo_typ						rt_info;
_LOCAL  UINT							CycleTime;

_LOCAL RTCtime_typ 						TimeBuf;

_LOCAL USINT 							Error;
_LOCAL UINT								idstat,brstate;

_LOCAL BOOL								initPAB;

_LOCAL_RETAIN Stats_Typ						SYS_Statistic	;

/*** eof *****************************************************************************/
```

#### iodrv_parse.h
```c
/******************************************************************************
*    COPYRIGHT    BERNECKER + RAINER Industrie-Elektronik Ges.m.b.H           *
*******************************************************************************
*  Projekt:  Protokoll Treiber IODRV (Profibus)
*  Teil:     Headerfile für Parser
*  Datei:    iodrv_parse.h
*  Typ:      GNU-C (32 Bit)
*------------------------------------------------------------------------------
*  Revision: 01.00
*  Datum:    05-04-2006
*  Autor:    WAI
*------------------------------------------------------------------------------
*  Funktion:
*------------------------------------------------------------------------------
*  Rev.  | Datum    | Name | Kommentar
*  ------+----------+------+---------------------------------------------------
*  01.00 | 05-04-06 | WAI  | Datei-Erstellung
*        |          |      |
******************************************************************************/
/***********************************************************************/
/* Konstantendefinition                                                */
/***********************************************************************/
#define ERR_MSG_PRE_STRG				"i/o"
#define MAX_ERROR_MSG_LOG				20				/* Anzahl Fehler, die in das Log-Buch eingetragen werden */

/* Bezeichnung der Datenmodule */
#define	DATA_OBJEKT_DPLIST				"dplist"
#define	DATA_OBJEKT_TYPLIST				"typlist"

/*-------------------------------------------------------
	Basisdatentypen
---------------------------------------------------------*/

#define BOOL_TYP						"_BOOL"
#define BOOL_IDX						0
#define USINT_TYP						"_USINT"
#define USINT_IDX						1
#define SINT_TYP						"_SINT"
#define SINT_IDX						2
#define UINT_TYP						"_UINT"
#define UINT_IDX						3
#define INT_TYP							"_INT"
#define INT_IDX							4
#define UDINT_TYP						"_UDINT"
#define UDINT_IDX						5
#define DINT_TYP						"_DINT"
#define DINT_IDX						6
#define REAL_TYP						"_REAL"
#define REAL_IDX						8

/*-------------------------------------------------------
	Fehlermeldungen
---------------------------------------------------------*/
#define NO_ERROR						0

/* Fehlermeldungen: Datenmodul nicht gefunden */
#define PARS_ERR_DPLIST_NOT_FOUND		501				/* Fehler: Datenmodul dplist nicht gefunden */
#define PARS_TXT_DPLIST_NOT_FOUND		"datamodule dplist not found"

#define PARS_ERR_TYPLIST_NOT_FOUND		502				/* Fehler: Datenmodul typlist nicht gefunden */
#define PARS_TXT_TYPLIST_NOT_FOUND		"datamodule typlist not found"

#define PARS_ERR_MEM_ALLOC				503				/* Fehler: Speicher kann nicht allokiert werden */
#define PARS_TXT_MEM_ALLOC				"TMP_alloc not successfull"

#define PARS_ERR_TO_MUCH_DEVICES		504				/* Fehler: Zuviele Geräte pro Linie angemeldet */
#define PARS_TXT_TO_MUCH_DEVICES		"to much devices for one line"

/* Fehlermeldungen des globalen Teiles */
#define PARS_ERR_UNKNOWN_GLOBAL_ENTRY	505				/* Fehler: Unbekannter Eintrag in globalen Bereich */
#define PARS_ERR_LINE_UNKNOWN			506				/* Fehler: Schnittstellendefinition kann keiner Linie zugeordnet werden */
#define PARS_ERR_TO_MUCH_LINES			507				/* Fehler: Anzahl deklarierter Linien zu gross (max. 6) */
#define PARS_ERR_NR_OF_LINES_ZERO		508				/* Fehler: Keine Linieneintraege im globalen Teil gefunden */
#define PARS_ERR_NR_OF_DP_ZERO			509				/* Fehler: Anzahl Datenpunkte einer Linie ist Null */
#define PARS_ERR_LINE_IF_NOT_DEFINED	510				/* Fehler: Einer Linie wurde keine Schnittstellenbeschreibung zugeordnet */
#define PARS_ERR_LINE_MODE_NOT_DEFINED	511				/* Fehler: Einer Linie wurde kein Schnittstellenmodus zugeordnet */
#define PARS_ERR_TIMEOUT_NOT_VALID		512				/* Fehler: Wert fuer Timeout ungueltig */
#define PARS_ERR_RETRY_ANZ_NOT_VALID	513				/* Fehler: Wert fuer Wiederholungen bei Telegrammfehlern ungueltig */
#define PARS_ERR_CONN_ANZ_NOT_VALID		514				/* Fehler: Wert fuer Anzahl Anmeldeversuche ungueltig */
#define PARS_ERR_WAIT_INTV_NOT_VALID	515				/* Fehler: Wert fuer Wartezeit für Anmeldeversuch ungueltig */
#define PARS_ERR_TIME_TS_NOT_VALID		516				/* Fehler: Wert fuer Zeitsyncronisation ungueltig */
#define PARS_ERR_IF_RESET_NOT_VALID		517				/* Fehler: Wert fuer Schnittstellen-Reset ungueltig */
#define PARS_ERR_TIME_CLASS2_NOT_VALID	518				/* Fehler: Wert fuer Abtastzeit Class 2 Telegramme ungueltig */
#define PARS_ERR_TIME_CLASS2F_NOT_VALID	519				/* Fehler: Wert fuer Hohe Abtastzeit Class 2 Telegramme ungueltig */
#define PARS_ERR_DD_ENABLE_NOT_VALID	520				/* Fehler: Wert fuer Freigabe Störschriebübertragung ungueltig */
#define PARS_ERR_DD_TIMEOUT_NOT_VALID	521				/* Fehler: Wert fuer Timeout Störschriebübertragung ungueltig */
#define PARS_ERR_DD_DELAY_NOT_VALID		522				/* Fehler: Wert fuer Verzögerung Störschriebübertragung ungueltig */
#define PARS_ERR_CMD_ENABLE_NOT_VALID	523				/* Fehler: Wert fuer Freigabe Kommandübertragung ungueltig */
#define PARS_ERR_CMD_TIMEOUT_NOT_VALID	524				/* Fehler: Wert fuer Timeout Kommandoübertragung ungueltig */

/* Fehlermeldungen des Datenpunktbereiches */
#define PARS_ERR_UNKNOWN_DP_ENTRY		600				/* Fehler: Unbekannter Eintrag in Datenpunkt Bereich */
#define PARS_ERR_ANLNR_NOT_DEFINED		601				/* Fehler: Anlagennummer nicht definiert */
#define PARS_ERR_DPNR_NOT_DEFINED		602				/* Fehler: Datenpunktnummer nicht definiert */
#define PARS_ERR_TYP_NOT_DEFINED		603				/* Fehler: Datentyp nicht definiert */
#define PARS_ERR_DPTYP_NR_NOT_DEFINED	609				/* Fehler: Datentyp Nummer nicht definiert */
#define PARS_ERR_ITEM_NR_NOT_DEFINED	610				/* Fehler: Item Nummer nicht definiert */
#define PARS_ERR_ITEM_TYP_NOT_DEFINED	611				/* Fehler: Item Typ nicht definiert */
#define PARS_ERR_ITEM_TYP_UNKNOWN		612				/* Fehler: Item Typ unbekannt */
#define PARS_ERR_ITEM_TYP_NOT_VALID		613				/* Fehler: Item Typ nicht gueltig (Analogwert->BOOL oder Doppelmeldung->BOOL) */
#define PARS_ERR_ITEM_NAME_NOT_DEFINED	614				/* Fehler: Item Typ nicht definiert */
#define PARS_ERR_IODRV_INV_NOT_DEFINED	615				/* Fehler: IODRV Invers nicht definiert */
#define PARS_ERR_IODRV_QUITT_NOT_DEFINED	616			/* Fehler: IODRV ReqTyp nicht definiert */
#define PARS_ERR_PV_NOT_FOUND			617				/* Fehler: IODRV PV nicht gefunden */

/* Fehlermeldungen des Itembereiches */
#define PARS_ERR_UNKNOWN_ITEM_ENTRY		700				/* Fehler: Unbekannter Eintrag in Item Bereich (DM typlist)*/

/*-------------------------------------------------------
	Schlüsselworte
---------------------------------------------------------*/
/* Hilfskonstanten */

#define ALL_SECTION						0				/* Es wird im allgemeinen Teil geparst (Meldungsunterdrückung) */
#define IODRV_SECTION						1				/* Es wird im IODRV - Teil geparst (Meldung bei unbekannten Schlüsselworten) */
#define DP_PART							0				/* Es wird im allgemeinen Datenpunktbereich geparst */
#define ITEM_PART						1				/* Es wird im allgemeinen Itembereich geparst */

/* Schluesselworte Sectionen */
#define	KW_IODRV_SECTION				"I/O"			/* Schlüsselwort für IODRV-Section */
#define	KW_ALL_SECTION					"ALL"			/* Schlüsselwort für Allgemeine-Section */
#define	KW_BRS_SECTION					"BRS"			/* Schlüsselwort für BRS-Section */
#define KW_ITEM_SECTION					"ITEM"			/* Schlüsselwort für ITEM-Section */
#define KW_BLOCK_SECTION				"BLOCK"			/* Schlüsswlwort für Blockdefinition */

/* Schluesselworte  globaler Teil */

/* Schluesselworte  Datenpunkt Teil */
#define KW_DP_ALL_ANL					"ANLAGE"		/* Schlüsselwort für Anlagennummer */
#define KW_DP_ALL_ANL_NR				"NR"			/* Schlüsselwort für Anlagennummer (ANLAGEN.NR) */
#define KW_DP_ALL_DP					"DP"			/* Schlüsselwort für Datenpunktnummer */
#define KW_DP_ALL_DP_NR					"NR"			/* Schlüsselwort für Datenpunktnummer (DP.NR) */
#define KW_DP_ALL_TYP					"TYP"			/* Schlüsselwort für Datenpunkttyp */
#define KW_DP_ALL_ITEM					"ITEM"			/* Schlüsselwort Item Datentyp */
#define KW_DP_ALL_ITEM_TYP				"TYP"			/* Schlüsselwort Item-Datentyp ITEM.TYP */
#define KW_DP_ALL_ITEM_NR				"NR"			/* Schlüsselwort Item-Nummer (ITEM.NR) */
#define KW_DP_ALL_ITEM_NAME				"NAME"			/* Schlüsselwort Item-Nummer (ITEM.NAME) */

/* Schlüsselworte TYPLIST	ALL-Teil Datenpunkt */
#define	KW_DPTYP_ALL_TYP				"TYP"			/* Schlüsselwort Datentyp Nummer */
#define KW_DPTYP_ALL_TYP_NR				"NR"			/* Schlüsselwort Datentyp Nummer (TYP.NR) */

/* Schlüsselworte TYPLIST	ALL-Teil ITEM */

#define KW_ITEM_ALL_ITEM_TYP			"TYP"			/* Schlüsselwort Item Datentyp */
#define KW_ITEM_ALL_ITEM				"ITEM"			/* Schlüsselwort Item-Nummer */
#define KW_ITEM_ALL_ITEM_NR				"NR"			/* Schlüsselwort Item-Nummer (ITEM.NR) */

/* Schlüsselworte TYPLIST	IODRV-Teil */
#define KW_ITEM_IODRV_INV				"INV"			/* Schlüsselwort für Invers */
#define	KW_ITEM_IODRV_QUITT				"QUITT"			/* Schlüsselwort für Quittierpflichtig */
#define	KW_ITEM_IODRV_DIR				"DIR"			/* Schlüsselwort für Schribrichtung R/W/RW */

/* Schlüsselworte TYPLIST	IODRV Teil für DIR */
#define KW_ITEM_IODRV_DIR_R				"R"				/* Schlüsselwort für Read */
#define cKW_READ						0
#define KW_ITEM_IODRV_DIR_W				"W"				/* Schlüsselwort für Write */
#define cKW_WRITE						1
#define KW_ITEM_IODRV_DIR_RW			"RW"			/* Schlüsselwort für ReadWrite */
#define cKW_READWRITE					2

/*-------------------------------------------------------
	Grenzwerte
---------------------------------------------------------*/

/* Grenzwerte der globalen Parameter */

#define IF_RESET_MIN					0				/* Minimaler Wert für Freigabe IF Reset (IF.RESET) */
#define IF_RESET_MAX					1				/* Maximaler Wert für Freigabe IF Reset (IF.RESET) */
#define TIMEOUT_MIN						10				/* Minimaler Wert fuer Timeout (TIMEOUT) (in ms) */
#define TIMEOUT_MAX						10000			/* Maximaler Wert fuer Timeout (TIMEOUT) (in ms) */
#define RETRY_ANZ_MIN					0				/* Minimaler Wert fuer Wiederholungen bei Telegrammfehlern (RETRY.ANZ) */
#define RETRY_ANZ_MAX					1000			/* Maximaler Wert fuer Wiederholungen bei Telegrammfehlern (RETRY.ANZ) */
#define CONN_ANZ_MIN					0				/* Minimaler Wert fuer Anzahl Anmeldeversuche (CONN.ANZ) */
#define CONN_ANZ_MAX					1000			/* Maximaler Wert fuer Anzahl Anmeldeversuche (CONN.ANZ) */
#define WAIT_INTV_MIN					0				/* Minimaler Wert fuer Wartezeit für Anmeldeversuch (WAIT.INTV) (in ms) */
#define WAIT_INTV_MAX					1000000			/* Maximaler Wert fuer Wartezeit für Anmeldeversuch (WAIT.INTV) (in ms) */
#define TIME_TS_MIN						0				/* Minimaler Wert fuer Zeitsyncronisation (TIME.TS) (in ms) */
#define TIME_TS_MAX						10000000		/* Maximaler Wert fuer Zeitsyncronisation (TIME.TS) (in ms) */
#define TIME_CLASS2_MIN					10				/* Minimaler Wert für Abtastzeit Class2 Telegramme (TIME.CLASS2) */
#define TIME_CLASS2_MAX					10000			/* Maximaler Wert für Abtastzeit Class2 Telegramme (TIME.CLASS2) */
#define TIME_CLASS2F_MIN				10				/* Minimaler Wert für hohe Abtastzeit Class2 Telegramme (TIME.CLASS2F) */
#define TIME_CLASS2F_MAX				10000			/* Maximaler Wert für hohe Abtastzeit Class2 Telegramme (TIME.CLASS2F) */
#define DD_ENABLE_MIN					0				/* Minimaler Wert für Freigabe der Störschriebübertragung (DD.ENABLE) */
#define DD_ENABLE_MAX					1				/* Maximaler Wert für Freigabe der Störschriebübertragung (DD.ENABLE) */
#define DD_TIMEOUT_MIN					1000			/* Minimaler Wert für Timeout bei Störschriebübertragung (DD.TIMEOUT) */
#define DD_TIMEOUT_MAX					500000			/* Maximaler Wert für hohe Abtastzeit Class2 Telegramme (DD.TIMEOUT) */
#define DD_DELAY_MIN					1000			/* Minimaler Wert für Verzögerung der Störschriebübertragung des gleichen Gerätes (DD.DELAY) */
#define DD_DELAY_MAX					500000			/* Maximaler Wert für Verzögerung der Störschriebübertragung des gleichen Gerätes (DD.DELAY) */
#define CMD_ENABLE_MIN					0				/* Minimaler Wert für Freigabe Kommandoübertragung (CMD.ENABLE) */
#define CMD_ENABLE_MAX					1				/* Maximaler Wert für Freigabe Kommandoübertragung (CMD.ENABLE) */
#define CMD_TIMEOUT_MIN					1000			/* Minimaler Wert für Timeout bei Kommandoübertragung (CMD.TIMEOUT) */
#define CMD_TIMEOUT_MAX					500000			/* Maximaler Wert für Timeout bei Kommandoübertragung (CMD.TIMEOUT) */

/* Grenzwerte der Datenpunkt Parameter */

#define DEV_ADR_MIN						1				/* Minimaler Wert fuer Device Adresse */
#define DEV_ADR_MAX						254				/* Maximaler Wert fuer Device Adresse */
#define IODRV_TYPE_MIN					0				/* Minimaler Wert fuer IODRV-Type */
#define IODRV_TYPE_MAX					255				/* Maximaler Wert fuer IODRV-Type */
#define IODRV_INFO_MIN					0				/* Minimaler Wert fuer IODRV-Info */
#define IODRV_INFO_MAX					255				/* Maximaler Wert fuer IODRV-Info */
#define IODRV_ANALOGNR_MIN				1				/* Minimaler Wert fuer IODRV-Analogwert Nr. */
#define IODRV_ANALOGNR_MAX				MAX_ANALOGWERTE	/* Maximaler Wert fuer IODRV-Analogwert Nr. */
#define RAW_MIN							-4096			/* Minimaler Wert fuer Normierung Rohwert */
#define RAW_MAX							4095			/* Maximaler Wert fuer Normierung Rohwert */
#define NORM_MIN						-2000000000		/* Minimaler Wert fuer Normierung Normierungswert */
#define NORM_MAX						2000000000		/* Maximaler Wert fuer Normierung Normierungswert */
#define TSYNCH_MIN						0				/* Minimaler Wert fuer Zeitsynchronisation ein/aus */
#define TSYNCH_MAX						1				/* Minimaler Wert fuer Zeitsynchronisation ein/aus */
#define MRUC_MIN						0				/* Minimaler Wert fuer Aktivierung der Rücksetzung über LED-Taste */
#define MRUC_MAX						1				/* Minimaler Wert fuer Aktivierung der Rücksetzung über LED-Taste */
#define MRUC_TYPE_MIN			IODRV_TYPE_MIN			/* Minimaler Wert fuer Type.Nr zur Aktivierung der Rücksetzung über LED-Taste */
#define MRUC_TYPE_MAX			IODRV_TYPE_MAX			/* Minimaler Wert fuer Type.Nr zur Aktivierung der Rücksetzung über LED-Taste */
#define MRUC_INFO_MIN			IODRV_INFO_MIN			/* Minimaler Wert fuer Info.Nr zur Aktivierung der Rücksetzung über LED-Taste */
#define MRUC_INFO_MAX			IODRV_INFO_MAX			/* Minimaler Wert fuer Info.Nr zur Aktivierung der Rücksetzung über LED-Taste */
#define MODE_MIN						0				/* Minimaler Wert fuer Mode */
#define MODE_MAX						15				/* Maximaler Wert fuer Mode */

/***********************************************************************/
/* Datentypdeklaration                                                 */
/***********************************************************************/
typedef struct
{
	plcbit					defined;
	long					value;
} IODRV_ParserParInfo_typ;

typedef struct
{
	plcbit					defined;
	REAL					value;
} IODRV_ParserParRealInfo_typ;

typedef struct
{
	plcbit					defined;
	unsigned char			*name;
	unsigned short			size;
} IODRV_ParserTypInfo_typ;

/* --------------------------*/
/* Globale Parameter         */
/* --------------------------*/

typedef struct
{
	IODRV_ParserTypInfo_typ	Interface;
	IODRV_ParserParInfo_typ	LineNr;
} IODRV_GlobalLineData_typ;

typedef struct
{
	IODRV_ParserParInfo_typ	Dummy;
} IODRV_GlobalData_typ;

/* ----------------------------*/
/* Parameter Datenpunkt / Item */
/* ----------------------------*/

typedef struct
{
	IODRV_ParserParInfo_typ	AnlagenNr;
	IODRV_ParserParInfo_typ	DPNr;
	IODRV_ParserTypInfo_typ	Typ;
	IODRV_ParserParInfo_typ	DPTypNr;
	IODRV_ParserTypInfo_typ	DPName;
	IODRV_ParserParInfo_typ	ItemNr;
	IODRV_ParserTypInfo_typ	ItemTyp;
	IODRV_ParserParInfo_typ	ItemTypNr;
	IODRV_ParserTypInfo_typ	ItemName;
	IODRV_ParserParInfo_typ	Invers;
	IODRV_ParserParInfo_typ	Quitt;
	IODRV_ParserParInfo_typ	Dir;
} IODRV_ItemData_typ;

/* -----------------------------*/
/* Infos des Parsers			*/
/* -----------------------------*/

/* Infos des Parsers */
typedef struct
{
	unsigned short			NrOfDataPoints;
	unsigned short			NrOfItems;
	unsigned short			ActItemIdx;
	long					memAdr;
	long					memSize;
	unsigned short			allocStatus;
	plcbit					ErrorMsg;
	unsigned short			NrOfLogEntrys;
	unsigned short			error;
	unsigned short			warning;
} IODRV_ParserInfo_typ;

/* Hilfsvariable des Parsers */
typedef struct {
	unsigned char			*pParser;
	unsigned char			*pParserLine;
	unsigned char			*pParserErr;
	unsigned char			*pDataArg1;
	unsigned char			*pDataArg2;
	unsigned char			*pDataArg3;
	unsigned short			SizeArg1;
	unsigned short			SizeArg2;
	unsigned short			SizeArg3;
	unsigned short			SectionType;
	unsigned short			CountLines;
} Parser_typ;

typedef struct {
	plcbit					showData;
	plcbit					DataValid;
	unsigned short			AnlagenNr;
	unsigned short			DPTypNr;
	unsigned short			DPNr;
	unsigned short			ItemNr;
	IODRV_DP_Info_typ 		*pItemData;
	unsigned short			ItemIdx;
} IODRV_ItemDiagnose_typ;

/***********************************************************************/
/* Prototypen		                                                   */
/***********************************************************************/
void			iodrv_parser();
void			iodrv_parser_dplist_clear();
void			iodrv_parser_typlist_clear();
void			iodrv_parser_global();
void			iodrv_parser_dpinfo(plcbit *pBlockFound, plcbit *pDPFound);
unsigned short	get_line_idx(IODRV_ItemData_typ *pDPInfo, IODRV_GlobalData_typ *pGlobalData, unsigned short *LineIdx);
unsigned short	get_device_idx(unsigned short LineIdx, long DeviceAdr, unsigned short *DeviceIdx, plcbit *NewDevice);
plcbit			normierung_defined(IODRV_ItemData_typ *pItemData);
plcbit			iodrv_parser_dpinfo_ok(IODRV_ItemData_typ *pData);
plcbit			iodrv_parser_dptype(unsigned char *pName, unsigned short size);
plcbit			iodrv_parser_iteminfo();
plcbit			iodrv_parser_iteminfo_ok(IODRV_ItemData_typ *pData);
void			iodrv_parser_data(unsigned char *pSrcStart,unsigned char *pSrcEnd, Parser_typ *pPa, IODRV_ItemData_typ *pData, unsigned char SektorInfo, unsigned char PartInfo);
void			copyItemData(IODRV_ItemData_typ *pItemDest, IODRV_ItemData_typ *pItemSrc);
unsigned char	IsANumber(unsigned char *pData);
void			iodrv_parser_warn(unsigned short errorNr, unsigned char *pTxtInfo, unsigned char *pTxt0, unsigned char *pTxt1, long info1, unsigned char *pTxt2, long info2, unsigned char *pTxt3, long info3);
void			iodrv_parser_err(unsigned short errorNr, unsigned char *pTxtInfo, unsigned char *pTxt0, unsigned char *pTxt1, long info1, unsigned char *pTxt2, long info2, unsigned char *pTxt3, long info3);
void			iodrv_mem_diagnose();

/**********************************************************
*				Lokale Variablen Declaration
**********************************************************/

_LOCAL	Parser_typ				PaDPList,PaDPListSave;
_LOCAL	Parser_typ				PaTypList,PaTypListSave;
_LOCAL	DatObjInfo_typ			DOI_dplist,DOI_typlist;
_LOCAL	IODRV_ParserInfo_typ		IODRV_ParserInfo;
_LOCAL	IODRV_GlobalData_typ		IODRV_GlobalData;
_LOCAL	IODRV_ItemData_typ		IODRV_DPData,IODRV_ItemData,IODRV_BlockData;
_LOCAL_RETAIN	signed short			State_find_StationTypPoint, State_find_Section, State_find_Data	;
_LOCAL	unsigned char			MsgTxt[256];
_LOCAL	unsigned char			*pPointName;
_LOCAL	unsigned short			lenPointName;

#define ITEM_DIAGNOSE_SIZE		2
_LOCAL	IODRV_ItemDiagnose_typ	IODRV_ItemDiagnose[ITEM_DIAGNOSE_SIZE];
_LOCAL	IODRV_DP_Info_typ 		*pItemData0Diagnose;
_LOCAL	IODRV_DP_Info_typ 		*pItemData1Diagnose;

/*** eof *****************************************************************************/
```

- dbserv.h (reference to Logical/GlobalIncludes/dbserv.h)

- parser.h (reference to Logical/GlobalIncludes/parser.h)

- bksys.h (reference to Logical/GlobalIncludes/bksys.h)

- platform.h (reference to Logical/GlobalIncludes/platform.h)

### Program Logical/IO-Treiber/io (ANSIC, version 6.40.0) - Deklarartion der IO-Treiber-Variablen

#### io.c
```c
#ifdef _DEFAULT_INCLUDES
	#include <AsDefault.h>
#endif
#include <bur/plctypes.h>

/* Definition der I/O-Treiber-Variablen */

_GLOBAL BOOL IO_014001_GSx01100ASM03;
_GLOBAL BOOL IO_014001_GSx01100ASM05;
_GLOBAL BOOL IO_014001_GSx01100ASM06;
_GLOBAL BOOL IO_014001_GSx01100ASM07;
_GLOBAL BOOL IO_014001_GSx01100ASM08;
_GLOBAL BOOL IO_014001_GSx01100ASM09;
_GLOBAL BOOL IO_014001_GSx01100ASM31;
_GLOBAL BOOL IO_014001_GSx01100ASM32;
_GLOBAL BOOL IO_014001_GSx01100ASM33;
_GLOBAL BOOL IO_014001_GSx01100ASM34;
_GLOBAL BOOL IO_014001_GSx01100ABM01;
_GLOBAL BOOL IO_014001_GSx01100ABM07;
_GLOBAL BOOL IO_014001_GSx01100AGM02;
_GLOBAL BOOL IO_014001_GSx01100AGM03;

void _INIT init_io(void)
{
	IO_014001_GSx01100ASM03 = IO_014001_GSx01100ASM03;
	IO_014001_GSx01100ASM05 = IO_014001_GSx01100ASM05;
	IO_014001_GSx01100ASM06 = IO_014001_GSx01100ASM06;
	IO_014001_GSx01100ASM07 = IO_014001_GSx01100ASM07;
	IO_014001_GSx01100ASM08 = IO_014001_GSx01100ASM08;
	IO_014001_GSx01100ASM09 = IO_014001_GSx01100ASM09;
	IO_014001_GSx01100ASM31 = IO_014001_GSx01100ASM31;
	IO_014001_GSx01100ASM32 = IO_014001_GSx01100ASM32;
	IO_014001_GSx01100ASM33 = IO_014001_GSx01100ASM33;
	IO_014001_GSx01100ASM34 = IO_014001_GSx01100ASM34;
	IO_014001_GSx01100ABM01 = IO_014001_GSx01100ABM01;
	IO_014001_GSx01100ABM07 = IO_014001_GSx01100ABM07;
	IO_014001_GSx01100AGM02 = IO_014001_GSx01100AGM02;
	IO_014001_GSx01100AGM03 = IO_014001_GSx01100AGM03;

}

void _CYCLIC cyclic_io(void)
{
}
```

### Program Logical/Anwendung/kupplung (IEC, version 0.00.0) - Rangierung Kupplung SS2 von UMG SS1

#### kupplungCyclic.ld
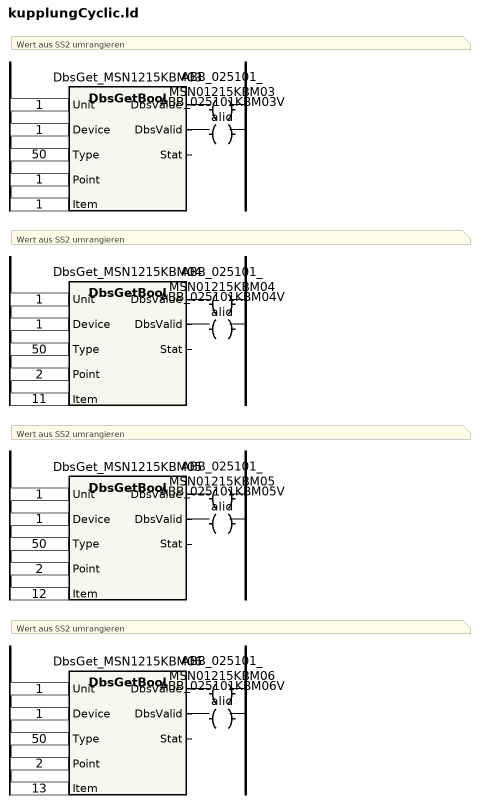
Diagram, in the editor's own instruction-list form stored in the file:
```il
PROGRAM _CYCLIC

{NetworkNumber := 1}
(* Wert aus SS2 umrangieren *)
LD	1
ST	DbsGet_MSN1215KBM03.Unit
LD	1
ST	DbsGet_MSN1215KBM03.Device
LD	50
ST	DbsGet_MSN1215KBM03.Type
LD	1
ST	DbsGet_MSN1215KBM03.Point
LD	1
ST	DbsGet_MSN1215KBM03.Item
CAL	DbsGet_MSN1215KBM03
LD	DbsGet_MSN1215KBM03.DbsValue
ST	ABB_025101_MSN01215KBM03
LD	DbsGet_MSN1215KBM03.DbsValid
ST	ABB_025101KBM03Valid

{NetworkNumber := 2}
(* Wert aus SS2 umrangieren *)
LD	1
ST	DbsGet_MSN1215KBM04.Unit
LD	1
ST	DbsGet_MSN1215KBM04.Device
LD	50
ST	DbsGet_MSN1215KBM04.Type
LD	2
ST	DbsGet_MSN1215KBM04.Point
LD	11
ST	DbsGet_MSN1215KBM04.Item
CAL	DbsGet_MSN1215KBM04
LD	DbsGet_MSN1215KBM04.DbsValue
ST	ABB_025101_MSN01215KBM04
LD	DbsGet_MSN1215KBM04.DbsValid
ST	ABB_025101KBM04Valid

{NetworkNumber := 3}
(* Wert aus SS2 umrangieren *)
LD	1
ST	DbsGet_MSN1215KBM05.Unit
LD	1
ST	DbsGet_MSN1215KBM05.Device
LD	50
ST	DbsGet_MSN1215KBM05.Type
LD	2
ST	DbsGet_MSN1215KBM05.Point
LD	12
ST	DbsGet_MSN1215KBM05.Item
CAL	DbsGet_MSN1215KBM05
LD	DbsGet_MSN1215KBM05.DbsValue
ST	ABB_025101_MSN01215KBM05
LD	DbsGet_MSN1215KBM05.DbsValid
ST	ABB_025101KBM05Valid

{NetworkNumber := 4}
(* Wert aus SS2 umrangieren *)
LD	1
ST	DbsGet_MSN1215KBM06.Unit
LD	1
ST	DbsGet_MSN1215KBM06.Device
LD	50
ST	DbsGet_MSN1215KBM06.Type
LD	2
ST	DbsGet_MSN1215KBM06.Point
LD	13
ST	DbsGet_MSN1215KBM06.Item
CAL	DbsGet_MSN1215KBM06
LD	DbsGet_MSN1215KBM06.DbsValue
ST	ABB_025101_MSN01215KBM06
LD	DbsGet_MSN1215KBM06.DbsValid
ST	ABB_025101KBM06Valid

END_PROGRAM
```

#### kupplungInit.ld
Diagram, in the editor's own instruction-list form stored in the file:
```il
PROGRAM _INIT

END_PROGRAM
```

#### kupplung.var
```iecst
VAR
	DbsGet_MSN1215KBM03 : DbsGetBool;
	DbsGet_MSN1215KBM04 : DbsGetBool;
	DbsGet_MSN1215KBM05 : DbsGetBool;
	DbsGet_MSN1215KBM06 : DbsGetBool;
	ABB_025101_MSN01215KBM03 : BOOL;
	ABB_025101KBM03Valid : BOOL;
	ABB_025101_MSN01215KBM04 : BOOL;
	ABB_025101KBM04Valid : BOOL;
	ABB_025101_MSN01215KBM05 : BOOL;
	ABB_025101KBM05Valid : BOOL;
	ABB_025101_MSN01215KBM06 : BOOL;
	ABB_025101KBM06Valid : BOOL;
END_VAR
```

### Data object Logical/Anwendung/dplist (Simple, version 0.00.0) - DbServ Datenpunktliste
